REGION Network 4: Генерация аварии
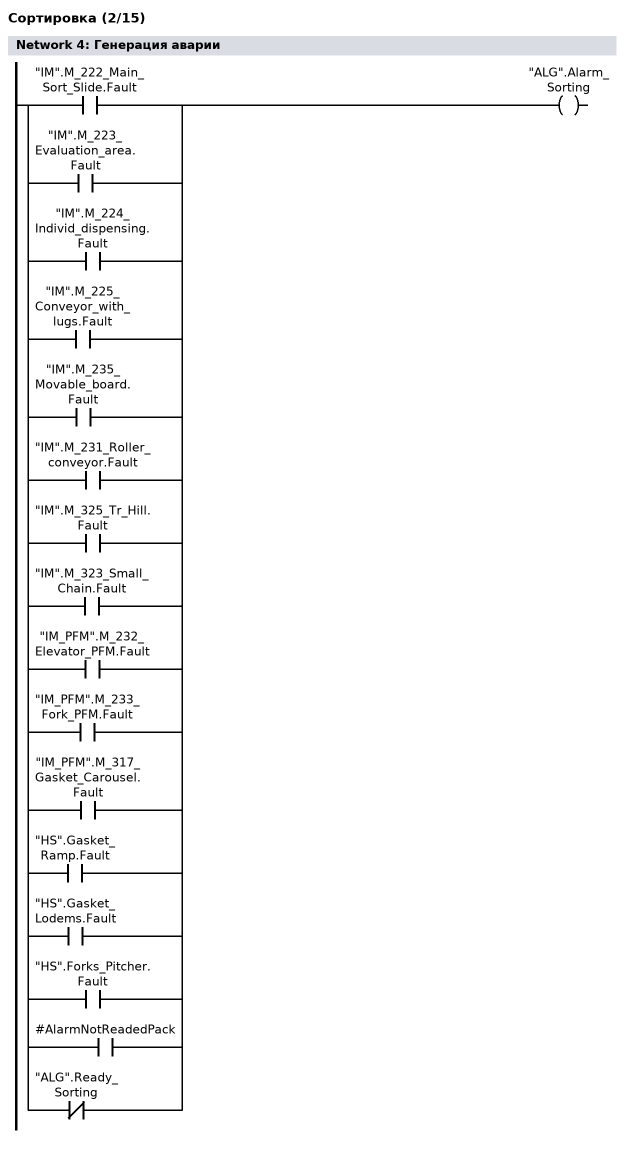
   RUNG wire#powerrail
      Contact( "IM".M_222_Main_Sort_Slide.Fault )
      wire#w1
      Coil( "ALG".Alarm_Sorting )
   END_RUNG
   RUNG wire#powerrail
      Contact( "IM".M_223_Evaluation_area.Fault )
   END_RUNG wire#w1
   RUNG wire#powerrail
      Contact( "IM".M_224_Individ_dispensing.Fault )
   END_RUNG wire#w1
   RUNG wire#powerrail
      Contact( "IM".M_225_Conveyor_with_lugs.Fault )
   END_RUNG wire#w1
   RUNG wire#powerrail
      Contact( "IM".M_235_Movable_board.Fault )
   END_RUNG wire#w1
   RUNG wire#powerrail
      Contact( "IM".M_231_Roller_conveyor.Fault )
   END_RUNG wire#w1
   RUNG wire#powerrail
      Contact( "IM".M_325_Tr_Hill.Fault )
   END_RUNG wire#w1
   RUNG wire#powerrail
      Contact( "IM".M_323_Small_Chain.Fault )
   END_RUNG wire#w1
   RUNG wire#powerrail
      Contact( "IM_PFM".M_232_Elevator_PFM.Fault )
   END_RUNG wire#w1
   RUNG wire#powerrail
      Contact( "IM_PFM".M_233_Fork_PFM.Fault )
   END_RUNG wire#w1
   RUNG wire#powerrail
      Contact( "IM_PFM".M_317_Gasket_Carousel.Fault )
   END_RUNG wire#w1
   RUNG wire#powerrail
      Contact( "HS".Gasket_Ramp.Fault )
   END_RUNG wire#w1
   RUNG wire#powerrail
      Contact( "HS".Gasket_Lodems.Fault )
   END_RUNG wire#w1
   RUNG wire#powerrail
      Contact( "HS".Forks_Pitcher.Fault )
   END_RUNG wire#w1
   RUNG wire#powerrail
      Contact( #AlarmNotReadedPack )
   END_RUNG wire#w1
   RUNG wire#powerrail
      I_Contact( "ALG".Ready_Sorting )
   END_RUNG wire#w1
   // the same network as SCL:
   "ALG".Alarm_Sorting := "IM".M_222_Main_Sort_Slide.Fault OR "IM".M_223_Evaluation_area.Fault OR "IM".M_224_Individ_dispensing.Fault OR "IM".M_225_Conveyor_with_lugs.Fault OR "IM".M_235_Movable_board.Fault OR "IM".M_231_Roller_conveyor.Fault OR "IM".M_325_Tr_Hill.Fault OR "IM".M_323_Small_Chain.Fault OR "IM_PFM".M_232_Elevator_PFM.Fault OR "IM_PFM".M_233_Fork_PFM.Fault OR "IM_PFM".M_317_Gasket_Carousel.Fault OR "HS".Gasket_Ramp.Fault OR "HS".Gasket_Lodems.Fault OR "HS".Forks_Pitcher.Fault OR #AlarmNotReadedPack OR NOT "ALG".Ready_Sorting;
END_REGION

REGION Network 5: Сбор аварий с других узлов + аварии не генерирующие останов линии
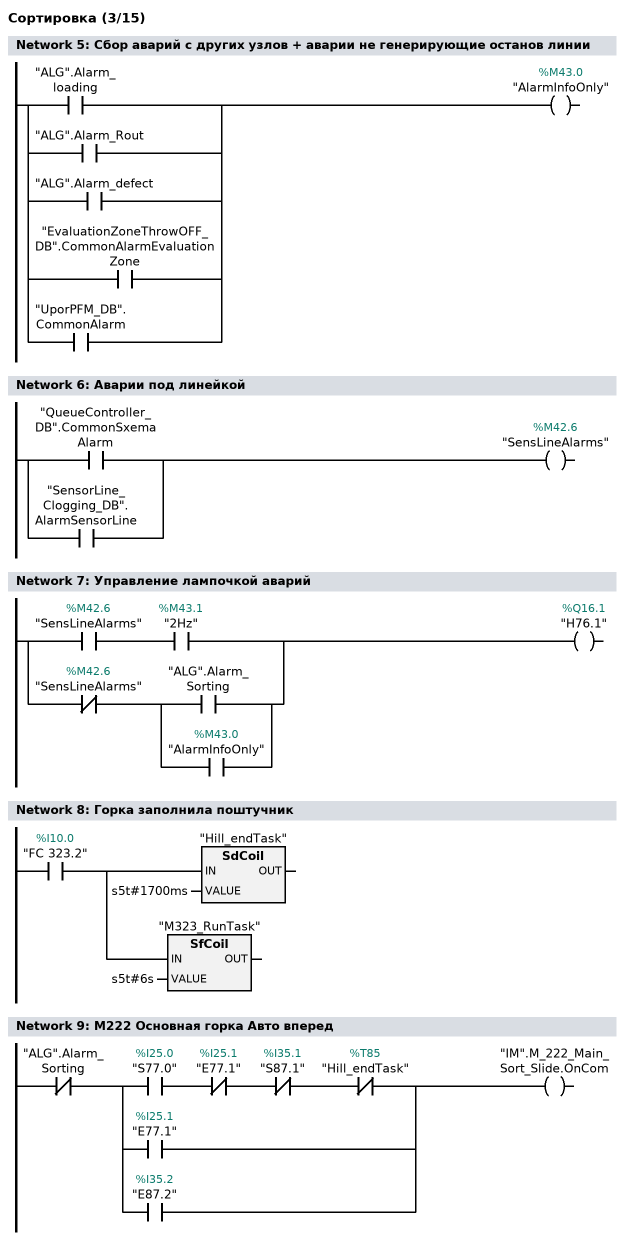
   RUNG wire#powerrail
      Contact( "ALG".Alarm_loading )
      wire#w1
      Coil( "AlarmInfoOnly" )
   END_RUNG
   RUNG wire#powerrail
      Contact( "ALG".Alarm_Rout )
   END_RUNG wire#w1
   RUNG wire#powerrail
      Contact( "ALG".Alarm_defect )
   END_RUNG wire#w1
   RUNG wire#powerrail
      Contact( "EvaluationZoneThrowOFF_DB".CommonAlarmEvaluationZone )
   END_RUNG wire#w1
   RUNG wire#powerrail
      Contact( "UporPFM_DB".CommonAlarm )
   END_RUNG wire#w1
   // the same network as SCL:
   "AlarmInfoOnly" := "ALG".Alarm_loading OR "ALG".Alarm_Rout OR "ALG".Alarm_defect OR "EvaluationZoneThrowOFF_DB".CommonAlarmEvaluationZone OR "UporPFM_DB".CommonAlarm;
END_REGION

REGION Network 6: Аварии под линейкой
   RUNG wire#powerrail
      Contact( "QueueController_DB".CommonSxemaAlarm )
      wire#w1
      Coil( "SensLineAlarms" )
   END_RUNG
   RUNG wire#powerrail
      Contact( "SensorLine_Clogging_DB".AlarmSensorLine )
   END_RUNG wire#w1
   // the same network as SCL:
   "SensLineAlarms" := "QueueController_DB".CommonSxemaAlarm OR "SensorLine_Clogging_DB".AlarmSensorLine;
END_REGION

REGION Network 7: Управление лампочкой аварий
   RUNG wire#powerrail
      Contact( "SensLineAlarms" )
      Contact( "2Hz" )
      wire#w1
      Coil( "H76.1" )
   END_RUNG
   RUNG wire#powerrail
      I_Contact( "SensLineAlarms" )
      wire#w2
      Contact( "ALG".Alarm_Sorting )
   END_RUNG wire#w1
   RUNG wire#w2
      Contact( "AlarmInfoOnly" )
   END_RUNG wire#w1
   // the same network as SCL:
   "H76.1" := ("SensLineAlarms" AND "2Hz") OR (NOT "SensLineAlarms" AND ("ALG".Alarm_Sorting OR "AlarmInfoOnly"));
END_REGION

REGION Network 8: Горка заполнила поштучник
   // no SCL statement known for SdCoil, SfCoil: written as a call
   #_w1 := "FC 323.2";
   SdCoil(in := "FC 323.2", value := s5t#1700ms, operand := "Hill_endTask");
   SfCoil(in := #_w1, value := s5t#6s, operand := "M323_RunTask");
END_REGION

REGION Network 9: М222 Основная горка Авто вперед
   RUNG wire#powerrail
      I_Contact( "ALG".Alarm_Sorting )
      wire#w1
      Contact( "S77.0" )
      I_Contact( "E77.1" )
      I_Contact( "S87.1" )
      I_Contact( "Hill_endTask" )
      wire#w2
      Coil( "IM".M_222_Main_Sort_Slide.OnCom )
   END_RUNG
   RUNG wire#w1
      Contact( "E77.1" )
   END_RUNG wire#w2
   RUNG wire#w1
      Contact( "E87.2" )
   END_RUNG wire#w2
   // the same network as SCL:
   "IM".M_222_Main_Sort_Slide.OnCom := NOT "ALG".Alarm_Sorting AND (("S77.0" AND NOT "E77.1" AND NOT "S87.1" AND NOT "Hill_endTask") OR "E77.1" OR "E87.2");
END_REGION

REGION Network 10: М222 Основная горка команда на движениее
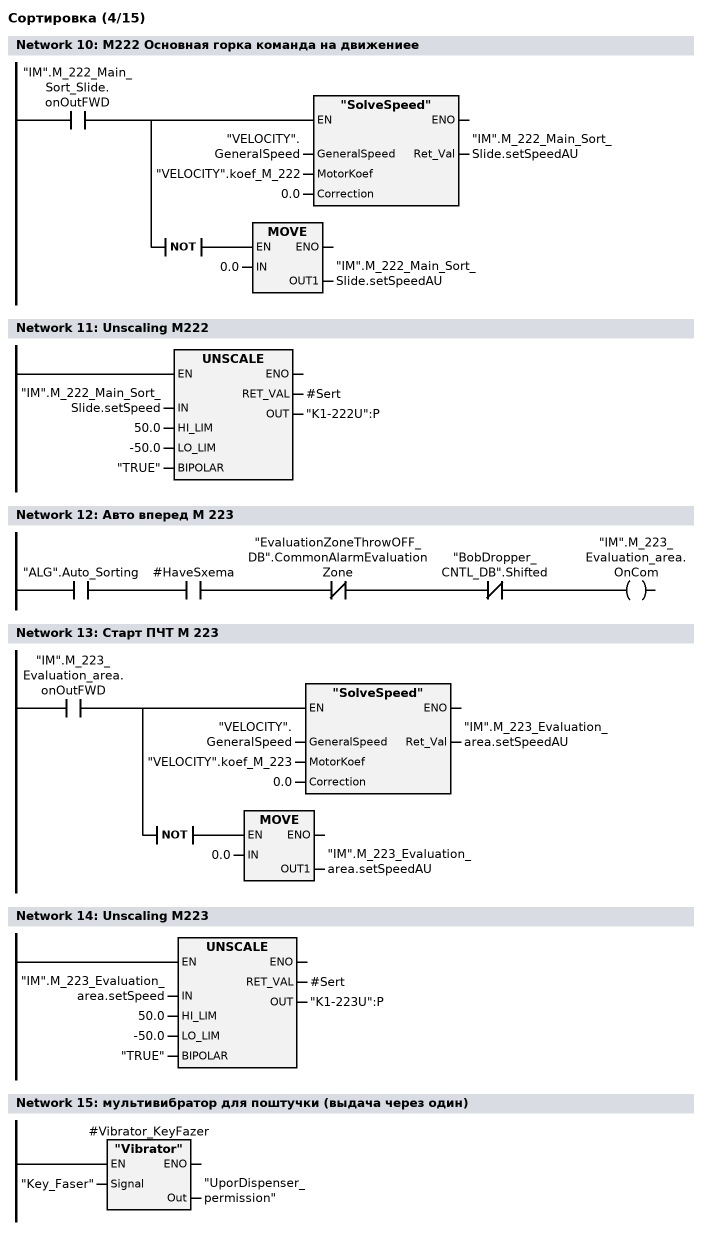
   RUNG wire#powerrail
      Contact( "IM".M_222_Main_Sort_Slide.onOutFWD )
      wire#w1
      "SolveSpeed"(GeneralSpeed := "VELOCITY".GeneralSpeed, MotorKoef := "VELOCITY".koef_M_222, Correction := 0.0, Ret_Val => "IM".M_222_Main_Sort_Slide.setSpeedAU)
   END_RUNG
   RUNG wire#w1
      Not()
      { S7_GenerateENO := "TRUE" } Move(in := 0.0, out1 => "IM".M_222_Main_Sort_Slide.setSpeedAU)
   END_RUNG
   // the same network as SCL:
   #_w1 := "IM".M_222_Main_Sort_Slide.onOutFWD;
   IF #_w1 THEN
       "IM".M_222_Main_Sort_Slide.setSpeedAU := "SolveSpeed"(GeneralSpeed := "VELOCITY".GeneralSpeed,
                               MotorKoef := "VELOCITY".koef_M_222,
                               Correction := 0.0);
   END_IF;
   IF NOT #_w1 THEN "IM".M_222_Main_Sort_Slide.setSpeedAU := 0.0; END_IF;
END_REGION

REGION Network 11: Unscaling M222
   RUNG wire#powerrail
      UNSCALE(IN := "IM".M_222_Main_Sort_Slide.setSpeed, HI_LIM := 50.0, LO_LIM := -50.0, BIPOLAR := "TRUE", RET_VAL => #Sert, OUT => "K1-222U":P)
   END_RUNG
   // the same network as SCL:
   #Sert := UNSCALE(IN := "IM".M_222_Main_Sort_Slide.setSpeed,
                    HI_LIM := 50.0,
                    LO_LIM := -50.0,
                    BIPOLAR := "TRUE",
                    OUT => "K1-222U":P);
END_REGION

REGION Network 12: Авто вперед M 223
   RUNG wire#powerrail
      Contact( "ALG".Auto_Sorting )
      Contact( #HaveSxema )
      I_Contact( "EvaluationZoneThrowOFF_DB".CommonAlarmEvaluationZone )
      I_Contact( "BobDropper_CNTL_DB".Shifted )
      Coil( "IM".M_223_Evaluation_area.OnCom )
   END_RUNG
   // the same network as SCL:
   "IM".M_223_Evaluation_area.OnCom := "ALG".Auto_Sorting AND #HaveSxema AND NOT "EvaluationZoneThrowOFF_DB".CommonAlarmEvaluationZone AND NOT "BobDropper_CNTL_DB".Shifted;
END_REGION

REGION Network 13: Старт ПЧТ М 223
   RUNG wire#powerrail
      Contact( "IM".M_223_Evaluation_area.onOutFWD )
      wire#w1
      "SolveSpeed"(GeneralSpeed := "VELOCITY".GeneralSpeed, MotorKoef := "VELOCITY".koef_M_223, Correction := 0.0, Ret_Val => "IM".M_223_Evaluation_area.setSpeedAU)
   END_RUNG
   RUNG wire#w1
      Not()
      { S7_GenerateENO := "TRUE" } Move(in := 0.0, out1 => "IM".M_223_Evaluation_area.setSpeedAU)
   END_RUNG
   // the same network as SCL:
   #_w1 := "IM".M_223_Evaluation_area.onOutFWD;
   IF #_w1 THEN
       "IM".M_223_Evaluation_area.setSpeedAU := "SolveSpeed"(GeneralSpeed := "VELOCITY".GeneralSpeed,
                               MotorKoef := "VELOCITY".koef_M_223,
                               Correction := 0.0);
   END_IF;
   IF NOT #_w1 THEN "IM".M_223_Evaluation_area.setSpeedAU := 0.0; END_IF;
END_REGION

REGION Network 14: Unscaling M223
   RUNG wire#powerrail
      UNSCALE(IN := "IM".M_223_Evaluation_area.setSpeed, HI_LIM := 50.0, LO_LIM := -50.0, BIPOLAR := "TRUE", RET_VAL => #Sert, OUT => "K1-223U":P)
   END_RUNG
   // the same network as SCL:
   #Sert := UNSCALE(IN := "IM".M_223_Evaluation_area.setSpeed,
                    HI_LIM := 50.0,
                    LO_LIM := -50.0,
                    BIPOLAR := "TRUE",
                    OUT => "K1-223U":P);
END_REGION

REGION Network 15: мультивибратор для поштучки (выдача через один)
   RUNG wire#powerrail
      #Vibrator_KeyFazer(Signal := "Key_Faser", Out => "UporDispenser_permission")
   END_RUNG
   // the same network as SCL:
   #Vibrator_KeyFazer(Signal := "Key_Faser", Out => "UporDispenser_permission");   // "Vibrator"
END_REGION

REGION Network 16: Есть схема для сортировки
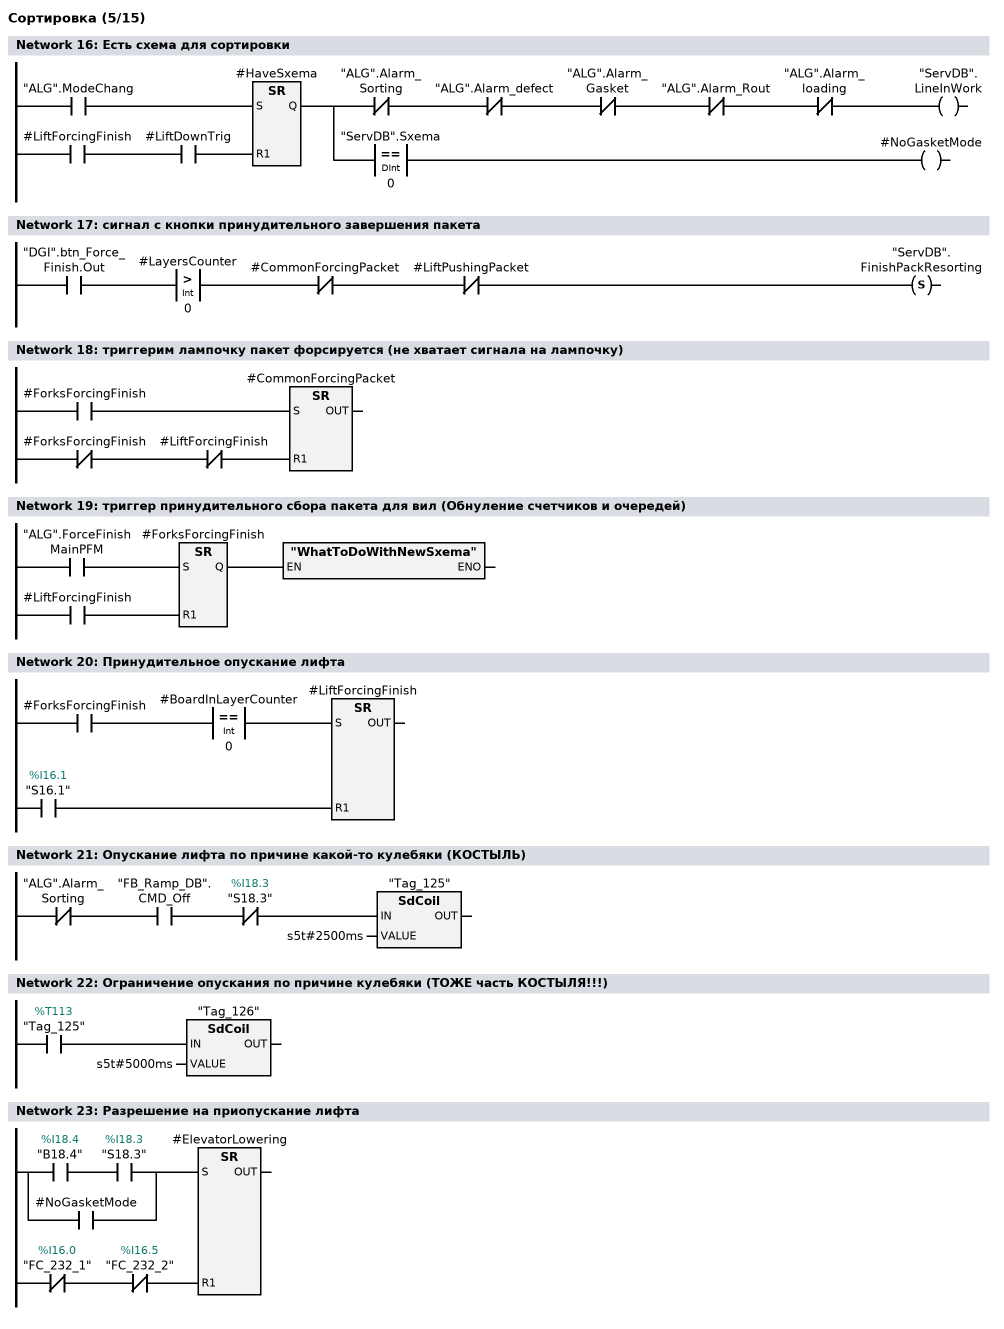
   RUNG wire#powerrail
      Contact( "ALG".ModeChang )
      S_SR(operand := #HaveSxema, r1 := wire#w1)
      wire#w2
      I_Contact( "ALG".Alarm_Sorting )
      I_Contact( "ALG".Alarm_defect )
      I_Contact( "ALG".Alarm_Gasket )
      I_Contact( "ALG".Alarm_Rout )
      I_Contact( "ALG".Alarm_loading )
      Coil( "ServDB".LineInWork )
   END_RUNG
   RUNG wire#powerrail
      Contact( #LiftForcingFinish )
      Contact( #LiftDownTrig )
   END_RUNG wire#w1
   RUNG wire#w2
      { S7_Templates := "SrcType := DInt" } EQ_Contact(in1 := "ServDB".Sxema, in2 := 0)
      Coil( #NoGasketMode )
   END_RUNG
   // the same network as SCL:
   IF "ALG".ModeChang THEN
       #HaveSxema := TRUE;   // SR flip-flop
   END_IF;
   IF #LiftForcingFinish AND #LiftDownTrig THEN #HaveSxema := FALSE; END_IF;
   "ServDB".LineInWork := #HaveSxema AND NOT "ALG".Alarm_Sorting AND NOT "ALG".Alarm_defect AND NOT "ALG".Alarm_Gasket AND NOT "ALG".Alarm_Rout AND NOT "ALG".Alarm_loading;
   #NoGasketMode := #HaveSxema AND ("ServDB".Sxema = 0);
END_REGION

REGION Network 17: сигнал с кнопки принудительного завершения пакета
   RUNG wire#powerrail
      Contact( "DGI".btn_Force_Finish.Out )
      { S7_Templates := "SrcType := Int" } GT_Contact(in1 := #LayersCounter, in2 := 0)
      I_Contact( #CommonForcingPacket )
      I_Contact( #LiftPushingPacket )
      S_Coil( "ServDB".FinishPackResorting )
   END_RUNG
   // the same network as SCL:
   IF "DGI".btn_Force_Finish.Out AND (#LayersCounter > 0) AND NOT #CommonForcingPacket AND NOT #LiftPushingPacket THEN
       "ServDB".FinishPackResorting := TRUE;
   END_IF;
END_REGION

REGION Network 18: триггерим лампочку пакет форсируется (не хватает сигнала на лампочку)
   RUNG wire#powerrail
      Contact( #ForksForcingFinish )
      S_SR(operand := #CommonForcingPacket, r1 := wire#w1)
   END_RUNG
   RUNG wire#powerrail
      I_Contact( #ForksForcingFinish )
      I_Contact( #LiftForcingFinish )
   END_RUNG wire#w1
   // the same network as SCL:
   IF #ForksForcingFinish THEN
       #CommonForcingPacket := TRUE;   // SR flip-flop
   END_IF;
   IF NOT #ForksForcingFinish AND NOT #LiftForcingFinish THEN #CommonForcingPacket := FALSE; END_IF;
END_REGION

REGION Network 19: триггер принудительного сбора пакета для вил (Обнуление счетчиков и очередей)
   RUNG wire#powerrail
      Contact( "ALG".ForceFinishMainPFM )
      S_SR(operand := #ForksForcingFinish, r1 := wire#w1)
      "WhatToDoWithNewSxema"()
   END_RUNG
   RUNG wire#powerrail
      Contact( #LiftForcingFinish )
   END_RUNG wire#w1
   // the same network as SCL:
   IF "ALG".ForceFinishMainPFM THEN
       #ForksForcingFinish := TRUE;   // SR flip-flop
   END_IF;
   IF #LiftForcingFinish THEN #ForksForcingFinish := FALSE; END_IF;
   IF #ForksForcingFinish THEN "WhatToDoWithNewSxema"(); END_IF;
END_REGION

REGION Network 20: Принудительное опускание лифта
   RUNG wire#powerrail
      Contact( #ForksForcingFinish )
      { S7_Templates := "SrcType := Int" } EQ_Contact(in1 := #BoardInLayerCounter, in2 := 0)
      S_SR(operand := #LiftForcingFinish, r1 := wire#w1)
   END_RUNG
   RUNG wire#powerrail
      Contact( "S16.1" )
   END_RUNG wire#w1
   // the same network as SCL:
   IF #ForksForcingFinish AND (#BoardInLayerCounter = 0) THEN
       #LiftForcingFinish := TRUE;   // SR flip-flop
   END_IF;
   IF "S16.1" THEN #LiftForcingFinish := FALSE; END_IF;
END_REGION

REGION Network 21: Опускание лифта по причине какой-то кулебяки (КОСТЫЛЬ)
   // no SCL statement known for SdCoil: written as a call
   SdCoil(in := NOT "ALG".Alarm_Sorting AND "FB_Ramp_DB".CMD_Off AND NOT "S18.3",
          value := s5t#2500ms,
          operand := "Tag_125");
END_REGION

REGION Network 22: Ограничение опускания по причине кулебяки (ТОЖЕ часть КОСТЫЛЯ!!!)
   // no SCL statement known for SdCoil: written as a call
   SdCoil(in := "Tag_125", value := s5t#5000ms, operand := "Tag_126");
END_REGION

REGION Network 23: Разрешение на приопускание лифта
   RUNG wire#powerrail
      Contact( "B18.4" )
      Contact( "S18.3" )
      wire#w1
      S_SR(operand := #ElevatorLowering, r1 := wire#w2)
   END_RUNG
   RUNG wire#powerrail
      Contact( #NoGasketMode )
   END_RUNG wire#w1
   RUNG wire#powerrail
      I_Contact( "FC_232_1" )
      I_Contact( "FC_232_2" )
   END_RUNG wire#w2
   // the same network as SCL:
   IF ("B18.4" AND "S18.3") OR #NoGasketMode THEN
       #ElevatorLowering := TRUE;   // SR flip-flop
   END_IF;
   IF NOT "FC_232_1" AND NOT "FC_232_2" THEN #ElevatorLowering := FALSE; END_IF;
END_REGION

REGION Network 24: Счёт слоёв
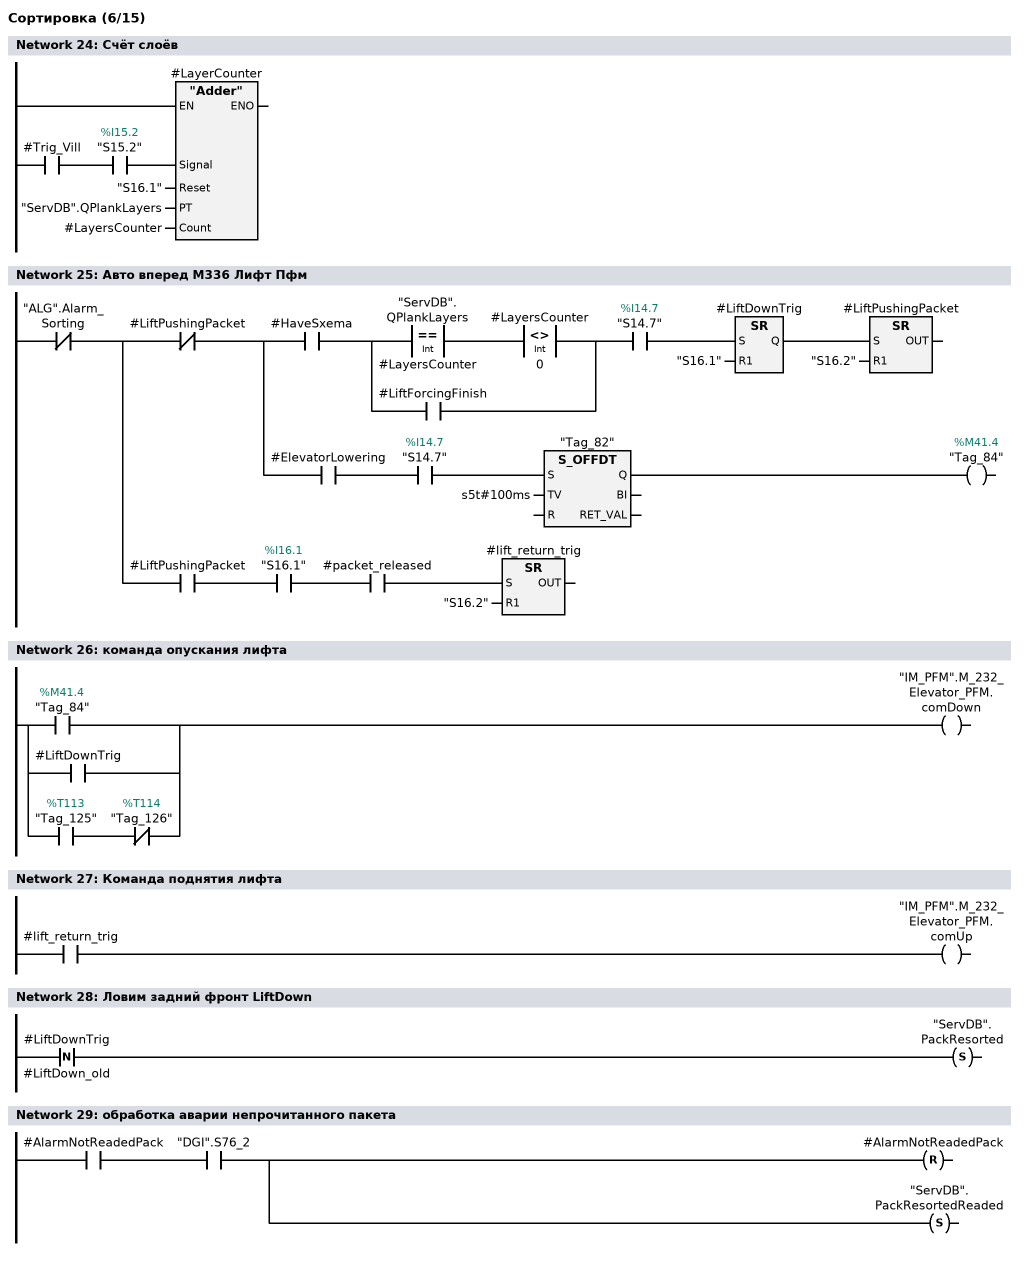
   RUNG wire#powerrail
      #LayerCounter(Signal := wire#w1, Reset := "S16.1", PT := "ServDB".QPlankLayers, Count := #LayersCounter)
   END_RUNG
   RUNG wire#powerrail
      Contact( #Trig_Vill )
      Contact( "S15.2" )
   END_RUNG wire#w1
   // the same network as SCL:
   #LayerCounter(Signal := #Trig_Vill AND "S15.2",   // "Adder"
                 Reset := "S16.1",
                 PT := "ServDB".QPlankLayers,
                 Count := #LayersCounter);
END_REGION

REGION Network 25: Авто вперед М336 Лифт Пфм
   RUNG wire#powerrail
      I_Contact( "ALG".Alarm_Sorting )
      wire#w1
      I_Contact( #LiftPushingPacket )
      wire#w2
      Contact( #HaveSxema )
      wire#w3
      { S7_Templates := "SrcType := Int" } EQ_Contact(in1 := "ServDB".QPlankLayers, in2 := #LayersCounter)
      { S7_Templates := "SrcType := Int" } NE_Contact(in1 := #LayersCounter, in2 := 0)
      wire#w4
      Contact( "S14.7" )
      S_SR(operand := #LiftDownTrig, r1 := "S16.1")
      S_SR(operand := #LiftPushingPacket, r1 := "S16.2")
   END_RUNG
   RUNG wire#w3
      Contact( #LiftForcingFinish )
   END_RUNG wire#w4
   RUNG wire#w2
      Contact( #ElevatorLowering )
      Contact( "S14.7" )
      S_OFFDT(T_NO := "Tag_82", TV := s5t#100ms, R :=, BI =>, RET_VAL =>)
      Coil( "Tag_84" )
   END_RUNG
   RUNG wire#w1
      Contact( #LiftPushingPacket )
      Contact( "S16.1" )
      Contact( #packet_released )
      S_SR(operand := #lift_return_trig, r1 := "S16.2")
   END_RUNG
   // the same network as SCL:
   #_w1 := NOT "ALG".Alarm_Sorting AND NOT #LiftPushingPacket;
   IF #_w1 AND #HaveSxema AND ((("ServDB".QPlankLayers = #LayersCounter) AND (#LayersCounter <> 0)) OR #LiftForcingFinish) AND "S14.7" THEN
       #LiftDownTrig := TRUE;   // SR flip-flop
   END_IF;
   IF "S16.1" THEN #LiftDownTrig := FALSE; END_IF;
   IF #LiftDownTrig THEN
       #LiftPushingPacket := TRUE;   // SR flip-flop
   END_IF;
   IF "S16.2" THEN #LiftPushingPacket := FALSE; END_IF;
   #_s5time1 := S_OFFDT(T_NO := "Tag_82",
                        S := #_w1 AND #ElevatorLowering AND "S14.7",
                        TV := s5t#100ms,
                        Q => #_w2);
   "Tag_84" := #_w2;
   IF NOT "ALG".Alarm_Sorting AND #LiftPushingPacket AND "S16.1" AND #packet_released THEN
       #lift_return_trig := TRUE;   // SR flip-flop
   END_IF;
   IF "S16.2" THEN #lift_return_trig := FALSE; END_IF;
END_REGION

REGION Network 26: команда опускания лифта
   RUNG wire#powerrail
      Contact( "Tag_84" )
      wire#w1
      Coil( "IM_PFM".M_232_Elevator_PFM.comDown )
   END_RUNG
   RUNG wire#powerrail
      Contact( #LiftDownTrig )
   END_RUNG wire#w1
   RUNG wire#powerrail
      Contact( "Tag_125" )
      I_Contact( "Tag_126" )
   END_RUNG wire#w1
   // the same network as SCL:
   "IM_PFM".M_232_Elevator_PFM.comDown := "Tag_84" OR #LiftDownTrig OR ("Tag_125" AND NOT "Tag_126");
END_REGION

REGION Network 27: Команда поднятия лифта
   RUNG wire#powerrail
      Contact( #lift_return_trig )
      Coil( "IM_PFM".M_232_Elevator_PFM.comUp )
   END_RUNG
   // the same network as SCL:
   "IM_PFM".M_232_Elevator_PFM.comUp := #lift_return_trig;
END_REGION

REGION Network 28: Ловим задний фронт LiftDown
   RUNG wire#powerrail
      N_Contact(operand := #LiftDownTrig, bit := #LiftDown_old)
      S_Coil( "ServDB".PackResorted )
   END_RUNG
   // the same network as SCL:
   #_w1 := NOT #LiftDownTrig AND #LiftDown_old;   // falling edge of #LiftDownTrig
   #LiftDown_old := #LiftDownTrig;
   IF #_w1 THEN "ServDB".PackResorted := TRUE; END_IF;
END_REGION

REGION Network 29: обработка аварии непрочитанного пакета
   RUNG wire#powerrail
      Contact( #AlarmNotReadedPack )
      Contact( "DGI".S76_2 )
      wire#w1
      R_Coil( #AlarmNotReadedPack )
   END_RUNG
   RUNG wire#w1
      S_Coil( "ServDB".PackResortedReaded )
   END_RUNG
   // the same network as SCL:
   #_w1 := #AlarmNotReadedPack AND "DGI".S76_2;
   IF #_w1 THEN
       #AlarmNotReadedPack := FALSE;
       "ServDB".PackResortedReaded := TRUE;
   END_IF;
END_REGION

REGION Network 30: Ловим задний фронт LiftPushing
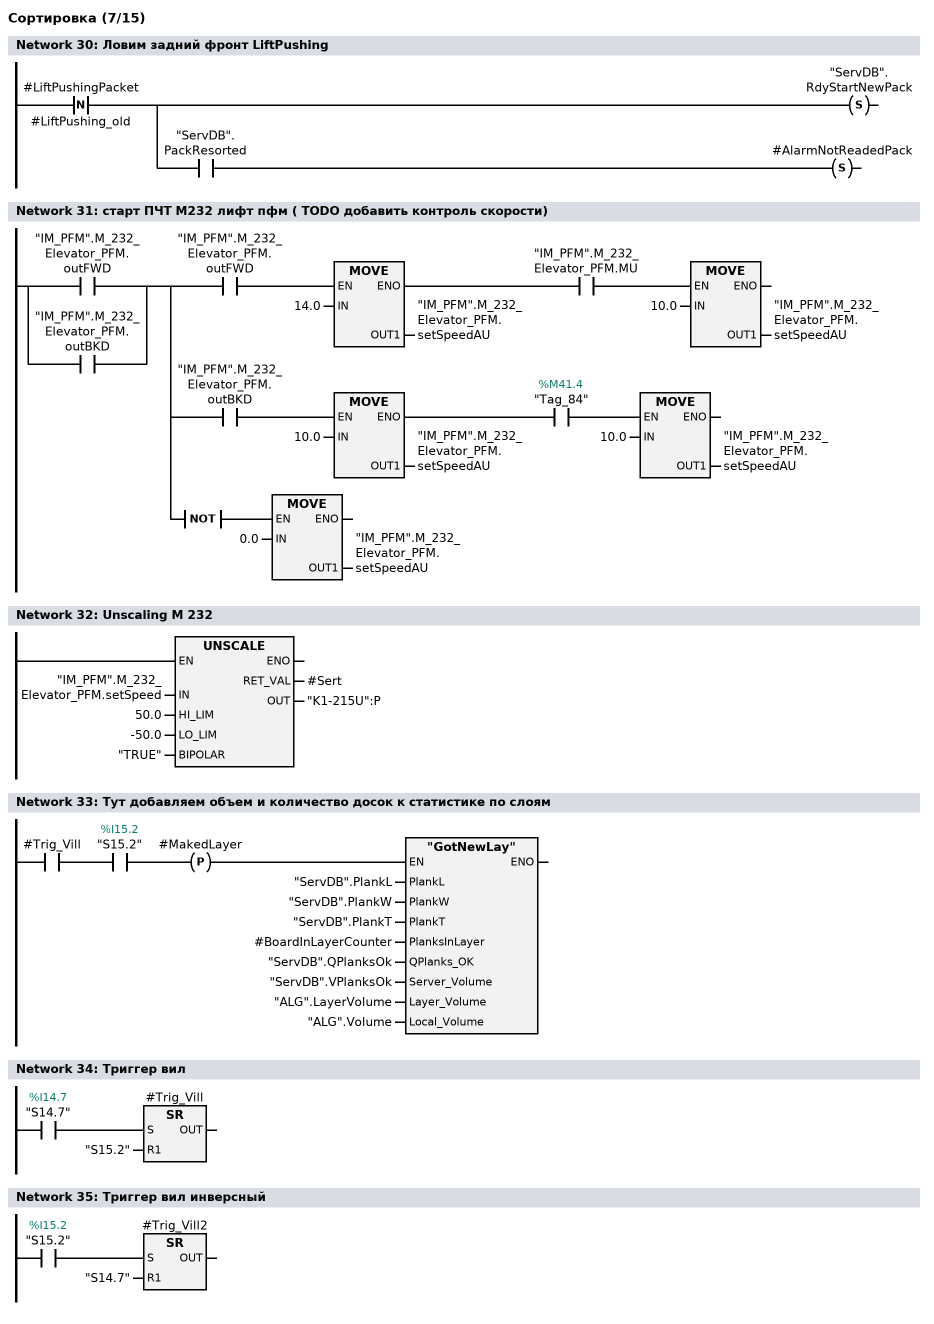
   RUNG wire#powerrail
      N_Contact(operand := #LiftPushingPacket, bit := #LiftPushing_old)
      wire#w1
      S_Coil( "ServDB".RdyStartNewPack )
   END_RUNG
   RUNG wire#w1
      Contact( "ServDB".PackResorted )
      S_Coil( #AlarmNotReadedPack )
   END_RUNG
   // the same network as SCL:
   #_w1 := NOT #LiftPushingPacket AND #LiftPushing_old;   // falling edge of #LiftPushingPacket
   #LiftPushing_old := #LiftPushingPacket;
   IF #_w1 THEN "ServDB".RdyStartNewPack := TRUE; END_IF;
   IF #_w1 AND "ServDB".PackResorted THEN #AlarmNotReadedPack := TRUE; END_IF;
END_REGION

REGION Network 31: старт ПЧТ М232 лифт пфм ( TODO добавить контроль скорости)
   RUNG wire#powerrail
      Contact( "IM_PFM".M_232_Elevator_PFM.outFWD )
      wire#w1
      Contact( "IM_PFM".M_232_Elevator_PFM.outFWD )
      { S7_GenerateENO := "TRUE" } Move(in := 14.0, out1 => "IM_PFM".M_232_Elevator_PFM.setSpeedAU)
      Contact( "IM_PFM".M_232_Elevator_PFM.MU )
      { S7_GenerateENO := "TRUE" } Move(in := 10.0, out1 => "IM_PFM".M_232_Elevator_PFM.setSpeedAU)
   END_RUNG
   RUNG wire#powerrail
      Contact( "IM_PFM".M_232_Elevator_PFM.outBKD )
   END_RUNG wire#w1
   RUNG wire#w1
      Contact( "IM_PFM".M_232_Elevator_PFM.outBKD )
      { S7_GenerateENO := "TRUE" } Move(in := 10.0, out1 => "IM_PFM".M_232_Elevator_PFM.setSpeedAU)
      Contact( "Tag_84" )
      { S7_GenerateENO := "TRUE" } Move(in := 10.0, out1 => "IM_PFM".M_232_Elevator_PFM.setSpeedAU)
   END_RUNG
   RUNG wire#w1
      Not()
      { S7_GenerateENO := "TRUE" } Move(in := 0.0, out1 => "IM_PFM".M_232_Elevator_PFM.setSpeedAU)
   END_RUNG
   // the same network as SCL:
   // ENO of a box is taken as its EN; it also drops when the box reports an error
   #_w1 := "IM_PFM".M_232_Elevator_PFM.outFWD OR "IM_PFM".M_232_Elevator_PFM.outBKD;
   #_w2 := #_w1 AND "IM_PFM".M_232_Elevator_PFM.outFWD;
   IF #_w2 THEN "IM_PFM".M_232_Elevator_PFM.setSpeedAU := 14.0; END_IF;
   IF #_w2 AND "IM_PFM".M_232_Elevator_PFM.MU THEN "IM_PFM".M_232_Elevator_PFM.setSpeedAU := 10.0; END_IF;
   #_w3 := #_w1 AND "IM_PFM".M_232_Elevator_PFM.outBKD;
   IF #_w3 THEN "IM_PFM".M_232_Elevator_PFM.setSpeedAU := 10.0; END_IF;
   IF #_w3 AND "Tag_84" THEN "IM_PFM".M_232_Elevator_PFM.setSpeedAU := 10.0; END_IF;
   IF NOT #_w1 THEN "IM_PFM".M_232_Elevator_PFM.setSpeedAU := 0.0; END_IF;
END_REGION

REGION Network 32: Unscaling M 232
   RUNG wire#powerrail
      UNSCALE(IN := "IM_PFM".M_232_Elevator_PFM.setSpeed, HI_LIM := 50.0, LO_LIM := -50.0, BIPOLAR := "TRUE", RET_VAL => #Sert, OUT => "K1-215U":P)
   END_RUNG
   // the same network as SCL:
   #Sert := UNSCALE(IN := "IM_PFM".M_232_Elevator_PFM.setSpeed,
                    HI_LIM := 50.0,
                    LO_LIM := -50.0,
                    BIPOLAR := "TRUE",
                    OUT => "K1-215U":P);
END_REGION

REGION Network 33: Тут добавляем объем и количество досок к статистике по слоям
   RUNG wire#powerrail
      Contact( #Trig_Vill )
      Contact( "S15.2" )
      P_Trig( #MakedLayer )
      "GotNewLay"(PlankL := "ServDB".PlankL, PlankW := "ServDB".PlankW, PlankT := "ServDB".PlankT, PlanksInLayer := #BoardInLayerCounter, QPlanks_OK := "ServDB".QPlanksOk, Server_Volume := "ServDB".VPlanksOk, Layer_Volume := "ALG".LayerVolume, Local_Volume := "ALG".Volume)
   END_RUNG
   // the same network as SCL:
   #_w1 := #Trig_Vill AND "S15.2";
   #_w2 := #_w1 AND NOT #MakedLayer;   // rising edge
   #MakedLayer := #_w1;
   IF #_w2 THEN
       "GotNewLay"(PlankL := "ServDB".PlankL,
                   PlankW := "ServDB".PlankW,
                   PlankT := "ServDB".PlankT,
                   PlanksInLayer := #BoardInLayerCounter,
                   QPlanks_OK := "ServDB".QPlanksOk,
                   Server_Volume := "ServDB".VPlanksOk,
                   Layer_Volume := "ALG".LayerVolume,
                   Local_Volume := "ALG".Volume);
   END_IF;
END_REGION

REGION Network 34: Триггер вил
   RUNG wire#powerrail
      Contact( "S14.7" )
      S_SR(operand := #Trig_Vill, r1 := "S15.2")
   END_RUNG
   // the same network as SCL:
   IF "S14.7" THEN
       #Trig_Vill := TRUE;   // SR flip-flop
   END_IF;
   IF "S15.2" THEN #Trig_Vill := FALSE; END_IF;
END_REGION

REGION Network 35: Триггер вил инверсный
   RUNG wire#powerrail
      Contact( "S15.2" )
      S_SR(operand := #Trig_Vill2, r1 := "S14.7")
   END_RUNG
   // the same network as SCL:
   IF "S15.2" THEN
       #Trig_Vill2 := TRUE;   // SR flip-flop
   END_IF;
   IF "S14.7" THEN #Trig_Vill2 := FALSE; END_IF;
END_REGION

REGION Network 36: Контроль кейфазеров на М225 и Счет досок на слой ПФМ (Счет не вызываем)
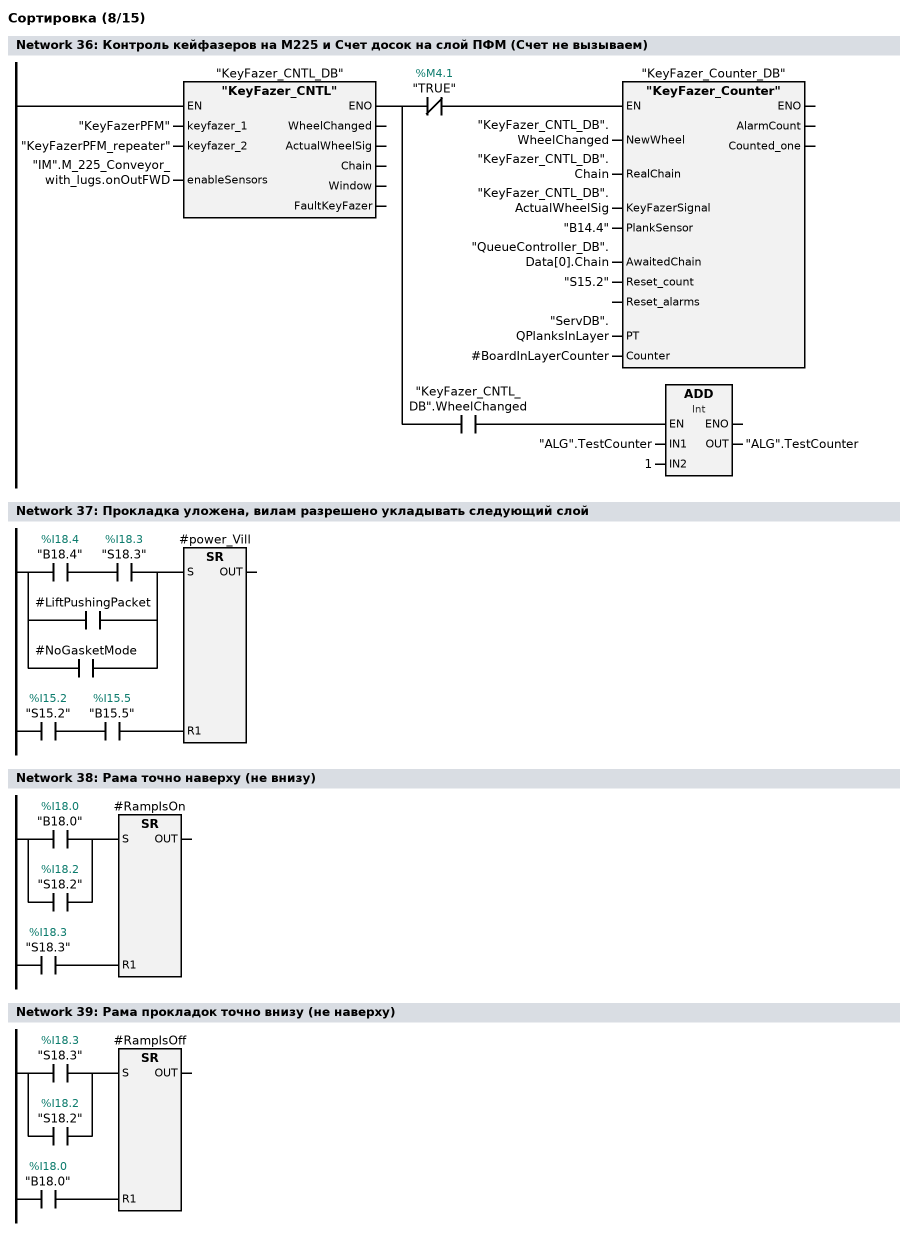
   RUNG wire#powerrail
      "KeyFazer_CNTL_DB"(keyfazer_1 := "KeyFazerPFM", keyfazer_2 := "KeyFazerPFM_repeater", enableSensors := "IM".M_225_Conveyor_with_lugs.onOutFWD, WheelChanged =>, ActualWheelSig =>, Chain =>, Window =>, FaultKeyFazer =>)
      wire#w1
      I_Contact( "TRUE" )
      "KeyFazer_Counter_DB"(NewWheel := "KeyFazer_CNTL_DB".WheelChanged, RealChain := "KeyFazer_CNTL_DB".Chain, KeyFazerSignal := "KeyFazer_CNTL_DB".ActualWheelSig, PlankSensor := "B14.4", AwaitedChain := "QueueController_DB".Data[0].Chain, Reset_count := "S15.2", Reset_alarms :=, PT := "ServDB".QPlanksInLayer, "Counter" := #BoardInLayerCounter, AlarmCount =>, Counted_one =>)
   END_RUNG
   RUNG wire#w1
      Contact( "KeyFazer_CNTL_DB".WheelChanged )
      { S7_Templates := "SrcType := Int"; S7_GenerateENO := "TRUE" } Add(in1 := "ALG".TestCounter, in2 := 1, out => "ALG".TestCounter)
   END_RUNG
   // the same network as SCL:
   "KeyFazer_CNTL_DB"(keyfazer_1 := "KeyFazerPFM",   // "KeyFazer_CNTL"
                      keyfazer_2 := "KeyFazerPFM_repeater",
                      enableSensors := "IM".M_225_Conveyor_with_lugs.onOutFWD,
                      ENO => #_w1);
   IF #_w1 AND NOT "TRUE" THEN
       "KeyFazer_Counter_DB"(NewWheel := "KeyFazer_CNTL_DB".WheelChanged,   // "KeyFazer_Counter"
                             RealChain := "KeyFazer_CNTL_DB".Chain,
                             KeyFazerSignal := "KeyFazer_CNTL_DB".ActualWheelSig,
                             PlankSensor := "B14.4",
                             AwaitedChain := "QueueController_DB".Data[0].Chain,
                             Reset_count := "S15.2",
                             PT := "ServDB".QPlanksInLayer,
                             "Counter" := #BoardInLayerCounter);
   END_IF;
   IF #_w1 AND "KeyFazer_CNTL_DB".WheelChanged THEN "ALG".TestCounter := "ALG".TestCounter + 1; END_IF;
END_REGION

REGION Network 37: Прокладка уложена, вилам разрешено укладывать следующий слой
   RUNG wire#powerrail
      Contact( "B18.4" )
      Contact( "S18.3" )
      wire#w1
      S_SR(operand := #power_Vill, r1 := wire#w2)
   END_RUNG
   RUNG wire#powerrail
      Contact( #LiftPushingPacket )
   END_RUNG wire#w1
   RUNG wire#powerrail
      Contact( #NoGasketMode )
   END_RUNG wire#w1
   RUNG wire#powerrail
      Contact( "S15.2" )
      Contact( "B15.5" )
   END_RUNG wire#w2
   // the same network as SCL:
   IF ("B18.4" AND "S18.3") OR #LiftPushingPacket OR #NoGasketMode THEN
       #power_Vill := TRUE;   // SR flip-flop
   END_IF;
   IF "S15.2" AND "B15.5" THEN #power_Vill := FALSE; END_IF;
END_REGION

REGION Network 38: Рама точно наверху (не внизу)
   RUNG wire#powerrail
      Contact( "B18.0" )
      wire#w1
      S_SR(operand := #RampIsOn, r1 := wire#w2)
   END_RUNG
   RUNG wire#powerrail
      Contact( "S18.2" )
   END_RUNG wire#w1
   RUNG wire#powerrail
      Contact( "S18.3" )
   END_RUNG wire#w2
   // the same network as SCL:
   IF "B18.0" OR "S18.2" THEN
       #RampIsOn := TRUE;   // SR flip-flop
   END_IF;
   IF "S18.3" THEN #RampIsOn := FALSE; END_IF;
END_REGION

REGION Network 39: Рама прокладок точно внизу (не наверху)
   RUNG wire#powerrail
      Contact( "S18.3" )
      wire#w1
      S_SR(operand := #RampIsOff, r1 := wire#w2)
   END_RUNG
   RUNG wire#powerrail
      Contact( "S18.2" )
   END_RUNG wire#w1
   RUNG wire#powerrail
      Contact( "B18.0" )
   END_RUNG wire#w2
   // the same network as SCL:
   IF "S18.3" OR "S18.2" THEN
       #RampIsOff := TRUE;   // SR flip-flop
   END_IF;
   IF "B18.0" THEN #RampIsOff := FALSE; END_IF;
END_REGION

REGION Network 40: M 233 вилы авто
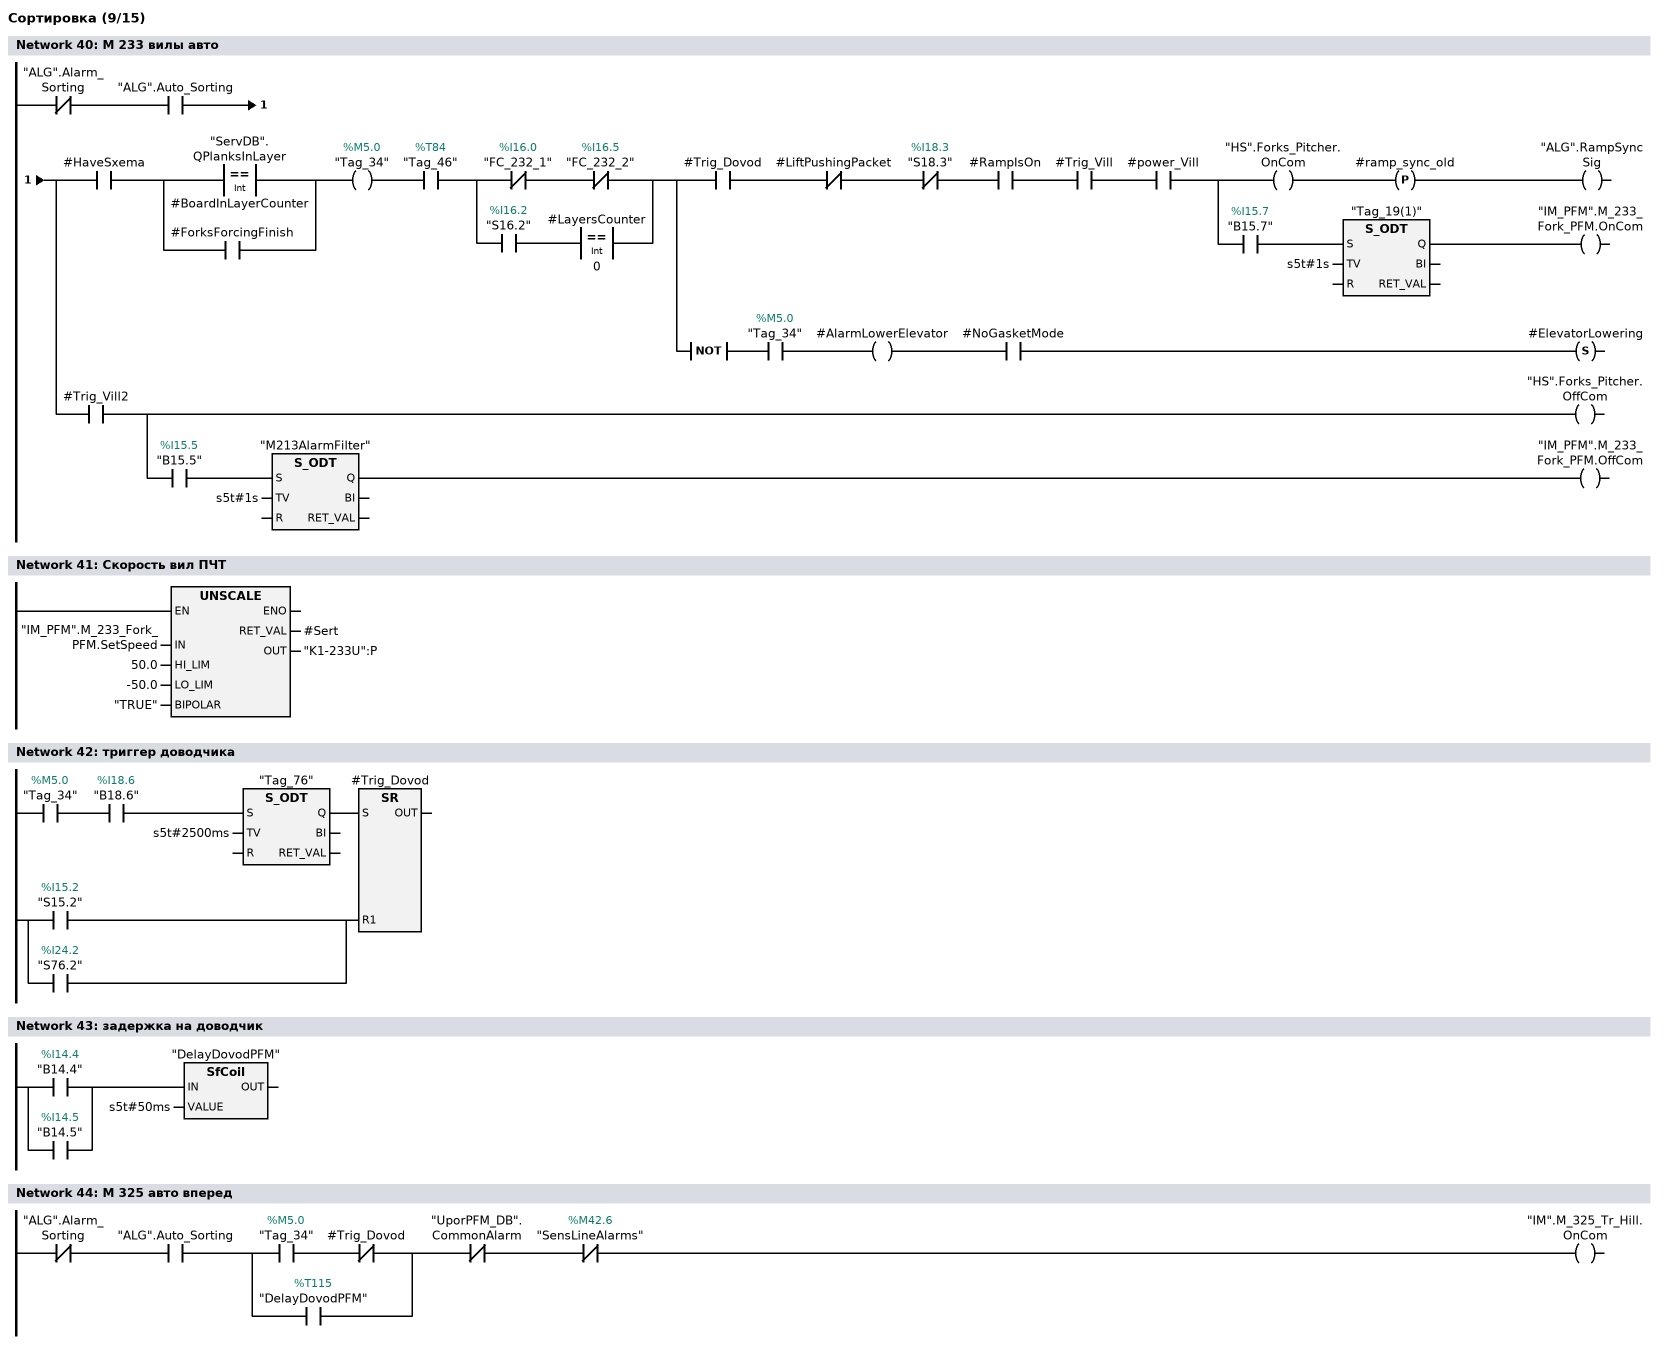
   RUNG wire#powerrail
      I_Contact( "ALG".Alarm_Sorting )
      Contact( "ALG".Auto_Sorting )
      wire#w1
      Contact( #HaveSxema )
      wire#w2
      { S7_Templates := "SrcType := Int" } EQ_Contact(in1 := "ServDB".QPlanksInLayer, in2 := #BoardInLayerCounter)
      wire#w3
      Coil( "Tag_34" )
      Contact( "Tag_46" )
      wire#w4
      I_Contact( "FC_232_1" )
      I_Contact( "FC_232_2" )
      wire#w5
      Contact( #Trig_Dovod )
      I_Contact( #LiftPushingPacket )
      I_Contact( "S18.3" )
      Contact( #RampIsOn )
      Contact( #Trig_Vill )
      Contact( #power_Vill )
      wire#w6
      Coil( "HS".Forks_Pitcher.OnCom )
      P_Trig( #ramp_sync_old )
      Coil( "ALG".RampSyncSig )
   END_RUNG
   RUNG wire#w2
      Contact( #ForksForcingFinish )
   END_RUNG wire#w3
   RUNG wire#w4
      Contact( "S16.2" )
      { S7_Templates := "SrcType := Int" } EQ_Contact(in1 := #LayersCounter, in2 := 0)
   END_RUNG wire#w5
   RUNG wire#w6
      Contact( "B15.7" )
      S_ODT(T_NO := "Tag_19(1)", TV := s5t#1s, R :=, BI =>, RET_VAL =>)
      Coil( "IM_PFM".M_233_Fork_PFM.OnCom )
   END_RUNG
   RUNG wire#w5
      Not()
      Contact( "Tag_34" )
      Coil( #AlarmLowerElevator )
      Contact( #NoGasketMode )
      S_Coil( #ElevatorLowering )
   END_RUNG
   RUNG wire#w1
      Contact( #Trig_Vill2 )
      wire#w7
      Coil( "HS".Forks_Pitcher.OffCom )
   END_RUNG
   RUNG wire#w7
      Contact( "B15.5" )
      S_ODT(T_NO := "M213AlarmFilter", TV := s5t#1s, R :=, BI =>, RET_VAL =>)
      Coil( "IM_PFM".M_233_Fork_PFM.OffCom )
   END_RUNG
   // the same network as SCL:
   #_w1 := NOT "ALG".Alarm_Sorting AND "ALG".Auto_Sorting;
   "Tag_34" := #_w1 AND #HaveSxema AND (("ServDB".QPlanksInLayer = #BoardInLayerCounter) OR #ForksForcingFinish);
   #_w2 := "Tag_34" AND "Tag_46" AND ((NOT "FC_232_1" AND NOT "FC_232_2") OR ("S16.2" AND (#LayersCounter = 0)));
   "HS".Forks_Pitcher.OnCom := #_w2 AND #Trig_Dovod AND NOT #LiftPushingPacket AND NOT "S18.3" AND #RampIsOn AND #Trig_Vill AND #power_Vill;
   #_w3 := "HS".Forks_Pitcher.OnCom AND NOT #ramp_sync_old;   // rising edge
   #ramp_sync_old := "HS".Forks_Pitcher.OnCom;
   "ALG".RampSyncSig := #_w3;
   #_s5time1 := S_ODT(T_NO := "Tag_19(1)", S := "HS".Forks_Pitcher.OnCom AND "B15.7", TV := s5t#1s, Q => #_w4);
   "IM_PFM".M_233_Fork_PFM.OnCom := #_w4;
   #AlarmLowerElevator := NOT #_w2 AND "Tag_34";
   IF #AlarmLowerElevator AND #NoGasketMode THEN #ElevatorLowering := TRUE; END_IF;
   "HS".Forks_Pitcher.OffCom := #_w1 AND #Trig_Vill2;
   #_s5time2 := S_ODT(T_NO := "M213AlarmFilter",
                      S := "HS".Forks_Pitcher.OffCom AND "B15.5",
                      TV := s5t#1s,
                      Q => #_w5);
   "IM_PFM".M_233_Fork_PFM.OffCom := #_w5;
END_REGION

REGION Network 41: Скорость вил ПЧТ
   RUNG wire#powerrail
      UNSCALE(IN := "IM_PFM".M_233_Fork_PFM.SetSpeed, HI_LIM := 50.0, LO_LIM := -50.0, BIPOLAR := "TRUE", RET_VAL => #Sert, OUT => "K1-233U":P)
   END_RUNG
   // the same network as SCL:
   #Sert := UNSCALE(IN := "IM_PFM".M_233_Fork_PFM.SetSpeed,
                    HI_LIM := 50.0,
                    LO_LIM := -50.0,
                    BIPOLAR := "TRUE",
                    OUT => "K1-233U":P);
END_REGION

REGION Network 42: триггер доводчика
   RUNG wire#powerrail
      Contact( "Tag_34" )
      Contact( "B18.6" )
      S_ODT(T_NO := "Tag_76", TV := s5t#2500ms, R :=, BI =>, RET_VAL =>)
      S_SR(operand := #Trig_Dovod, r1 := wire#w1)
   END_RUNG
   RUNG wire#powerrail
      Contact( "S15.2" )
   END_RUNG wire#w1
   RUNG wire#powerrail
      Contact( "S76.2" )
   END_RUNG wire#w1
   // the same network as SCL:
   #_s5time1 := S_ODT(T_NO := "Tag_76", S := "Tag_34" AND "B18.6", TV := s5t#2500ms, Q => #_w1);
   IF #_w1 THEN
       #Trig_Dovod := TRUE;   // SR flip-flop
   END_IF;
   IF "S15.2" OR "S76.2" THEN #Trig_Dovod := FALSE; END_IF;
END_REGION

REGION Network 43: задержка на доводчик
   // no SCL statement known for SfCoil: written as a call
   SfCoil(in := "B14.4" OR "B14.5", value := s5t#50ms, operand := "DelayDovodPFM");
END_REGION

REGION Network 44: M 325 авто вперед
   RUNG wire#powerrail
      I_Contact( "ALG".Alarm_Sorting )
      Contact( "ALG".Auto_Sorting )
      wire#w1
      Contact( "Tag_34" )
      I_Contact( #Trig_Dovod )
      wire#w2
      I_Contact( "UporPFM_DB".CommonAlarm )
      I_Contact( "SensLineAlarms" )
      Coil( "IM".M_325_Tr_Hill.OnCom )
   END_RUNG
   RUNG wire#w1
      Contact( "DelayDovodPFM" )
   END_RUNG wire#w2
   // the same network as SCL:
   "IM".M_325_Tr_Hill.OnCom := NOT "ALG".Alarm_Sorting AND "ALG".Auto_Sorting AND (("Tag_34" AND NOT #Trig_Dovod) OR "DelayDovodPFM") AND NOT "UporPFM_DB".CommonAlarm AND NOT "SensLineAlarms";
END_REGION

REGION Network 45: Старт ПЧТ 325
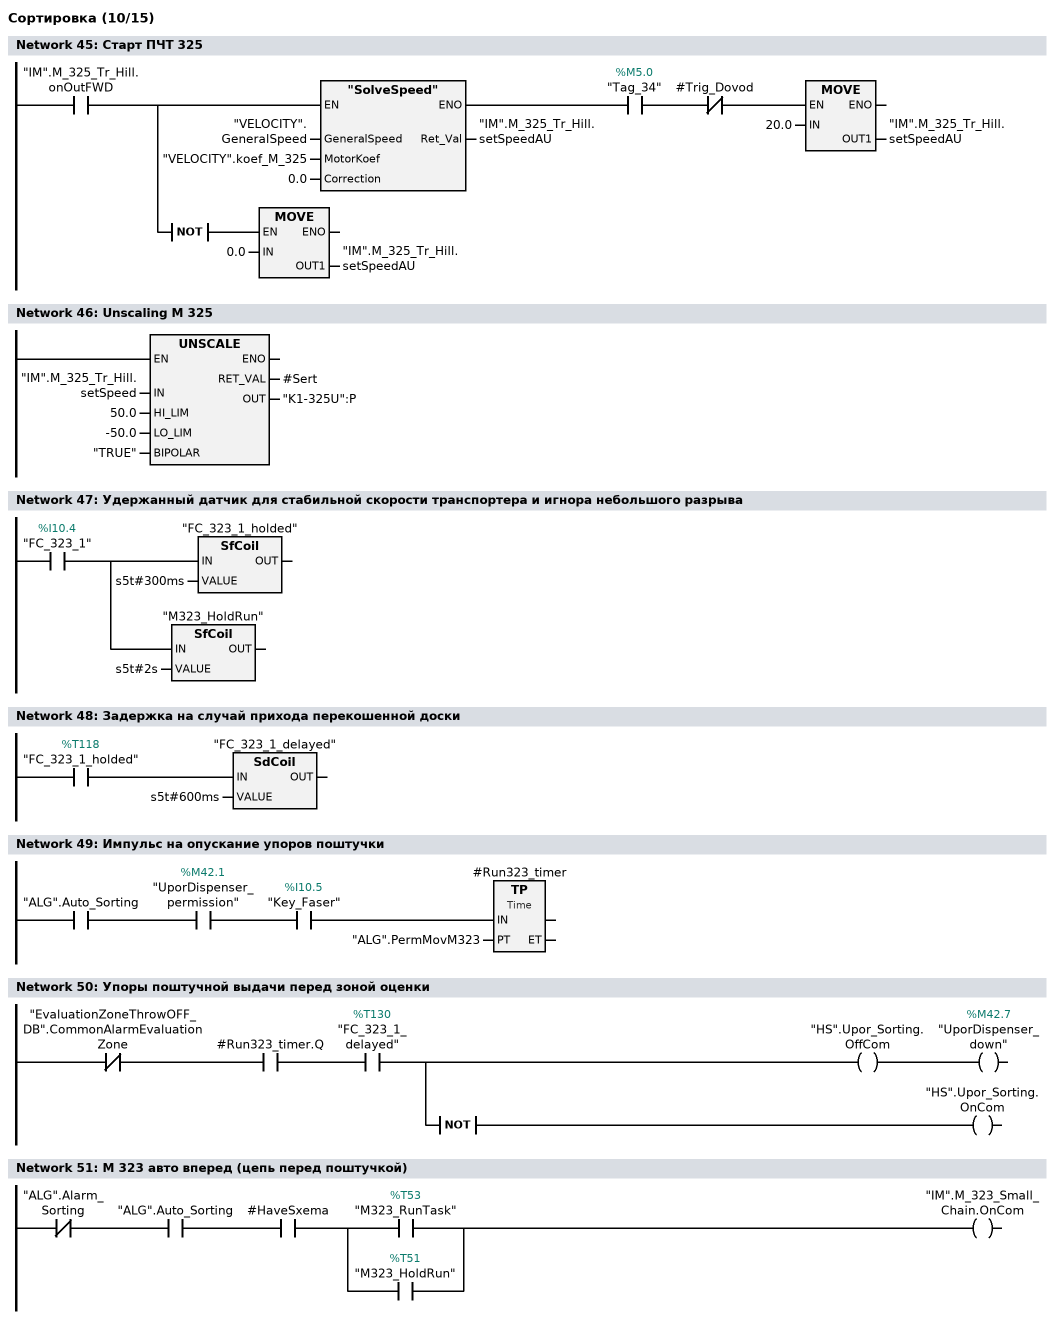
   RUNG wire#powerrail
      Contact( "IM".M_325_Tr_Hill.onOutFWD )
      wire#w1
      "SolveSpeed"(GeneralSpeed := "VELOCITY".GeneralSpeed, MotorKoef := "VELOCITY".koef_M_325, Correction := 0.0, Ret_Val => "IM".M_325_Tr_Hill.setSpeedAU)
      Contact( "Tag_34" )
      I_Contact( #Trig_Dovod )
      { S7_GenerateENO := "TRUE" } Move(in := 20.0, out1 => "IM".M_325_Tr_Hill.setSpeedAU)
   END_RUNG
   RUNG wire#w1
      Not()
      { S7_GenerateENO := "TRUE" } Move(in := 0.0, out1 => "IM".M_325_Tr_Hill.setSpeedAU)
   END_RUNG
   // the same network as SCL:
   #_w2 := "IM".M_325_Tr_Hill.onOutFWD;
   "IM".M_325_Tr_Hill.setSpeedAU := "SolveSpeed"(EN := "IM".M_325_Tr_Hill.onOutFWD,
                           GeneralSpeed := "VELOCITY".GeneralSpeed,
                           MotorKoef := "VELOCITY".koef_M_325,
                           Correction := 0.0,
                           ENO => #_w1);
   IF #_w1 AND "Tag_34" AND NOT #Trig_Dovod THEN "IM".M_325_Tr_Hill.setSpeedAU := 20.0; END_IF;
   IF NOT #_w2 THEN "IM".M_325_Tr_Hill.setSpeedAU := 0.0; END_IF;
END_REGION

REGION Network 46: Unscaling M 325
   RUNG wire#powerrail
      UNSCALE(IN := "IM".M_325_Tr_Hill.setSpeed, HI_LIM := 50.0, LO_LIM := -50.0, BIPOLAR := "TRUE", RET_VAL => #Sert, OUT => "K1-325U":P)
   END_RUNG
   // the same network as SCL:
   #Sert := UNSCALE(IN := "IM".M_325_Tr_Hill.setSpeed,
                    HI_LIM := 50.0,
                    LO_LIM := -50.0,
                    BIPOLAR := "TRUE",
                    OUT => "K1-325U":P);
END_REGION

REGION Network 47: Удержанный датчик для стабильной скорости транспортера и игнора небольшого разрыва
   // no SCL statement known for SfCoil: written as a call
   #_w1 := "FC_323_1";
   SfCoil(in := "FC_323_1", value := s5t#300ms, operand := "FC_323_1_holded");
   SfCoil(in := #_w1, value := s5t#2s, operand := "M323_HoldRun");
END_REGION

REGION Network 48: Задержка на случай прихода перекошенной доски
   // no SCL statement known for SdCoil: written as a call
   SdCoil(in := "FC_323_1_holded", value := s5t#600ms, operand := "FC_323_1_delayed");
END_REGION

REGION Network 49: Импульс на опускание упоров поштучки
   RUNG wire#powerrail
      Contact( "ALG".Auto_Sorting )
      Contact( "UporDispenser_permission" )
      Contact( "Key_Faser" )
      { S7_Templates := "time_type := Time" } #Run323_timer.TP(pt := "ALG".PermMovM323, et =>)
   END_RUNG
   // the same network as SCL:
   #Run323_timer.TP(IN := "ALG".Auto_Sorting AND "UporDispenser_permission" AND "Key_Faser",
                    PT := "ALG".PermMovM323);
END_REGION

REGION Network 50: Упоры поштучной выдачи перед зоной оценки
   RUNG wire#powerrail
      I_Contact( "EvaluationZoneThrowOFF_DB".CommonAlarmEvaluationZone )
      Contact( #Run323_timer.Q )
      Contact( "FC_323_1_delayed" )
      wire#w1
      Coil( "HS".Upor_Sorting.OffCom )
      Coil( "UporDispenser_down" )
   END_RUNG
   RUNG wire#w1
      Not()
      Coil( "HS".Upor_Sorting.OnCom )
   END_RUNG
   // the same network as SCL:
   "HS".Upor_Sorting.OffCom := NOT "EvaluationZoneThrowOFF_DB".CommonAlarmEvaluationZone AND #Run323_timer.Q AND "FC_323_1_delayed";
   "UporDispenser_down" := "HS".Upor_Sorting.OffCom;
   "HS".Upor_Sorting.OnCom := NOT "HS".Upor_Sorting.OffCom;
END_REGION

REGION Network 51: M 323 авто вперед (цепь перед поштучкой)
   RUNG wire#powerrail
      I_Contact( "ALG".Alarm_Sorting )
      Contact( "ALG".Auto_Sorting )
      Contact( #HaveSxema )
      wire#w1
      Contact( "M323_RunTask" )
      wire#w2
      Coil( "IM".M_323_Small_Chain.OnCom )
   END_RUNG
   RUNG wire#w1
      Contact( "M323_HoldRun" )
   END_RUNG wire#w2
   // the same network as SCL:
   "IM".M_323_Small_Chain.OnCom := NOT "ALG".Alarm_Sorting AND "ALG".Auto_Sorting AND #HaveSxema AND ("M323_RunTask" OR "M323_HoldRun");
END_REGION

REGION Network 52: Старт ПЧТ M 323
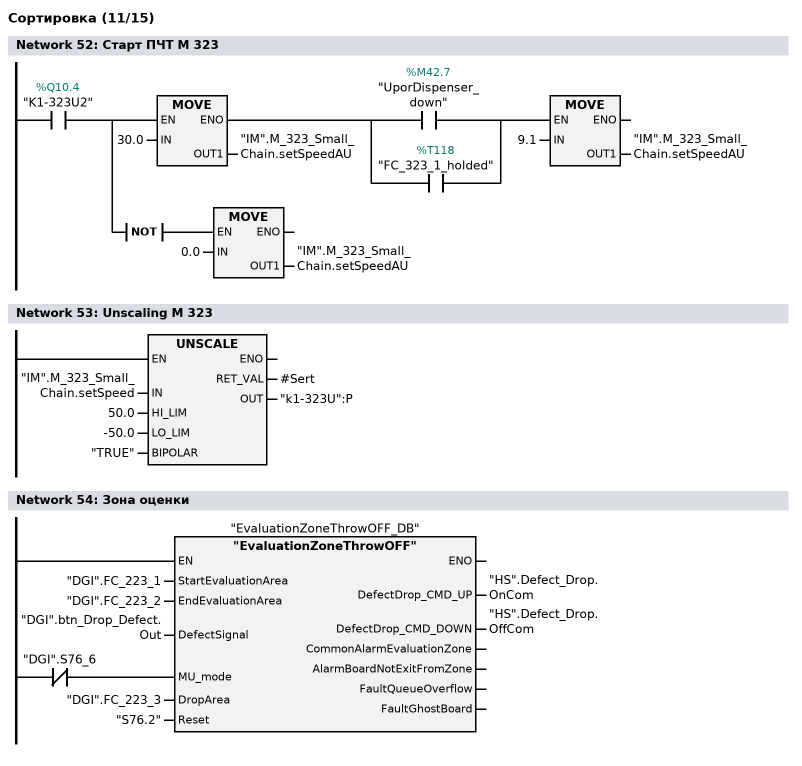
   RUNG wire#powerrail
      Contact( "K1-323U2" )
      wire#w1
      { S7_GenerateENO := "TRUE" } Move(in := 30.0, out1 => "IM".M_323_Small_Chain.setSpeedAU)
      wire#w2
      Contact( "UporDispenser_down" )
      wire#w3
      { S7_GenerateENO := "TRUE" } Move(in := 9.1, out1 => "IM".M_323_Small_Chain.setSpeedAU)
   END_RUNG
   RUNG wire#w2
      Contact( "FC_323_1_holded" )
   END_RUNG wire#w3
   RUNG wire#w1
      Not()
      { S7_GenerateENO := "TRUE" } Move(in := 0.0, out1 => "IM".M_323_Small_Chain.setSpeedAU)
   END_RUNG
   // the same network as SCL:
   // ENO of a box is taken as its EN; it also drops when the box reports an error
   IF "K1-323U2" THEN "IM".M_323_Small_Chain.setSpeedAU := 30.0; END_IF;
   IF "K1-323U2" AND ("UporDispenser_down" OR "FC_323_1_holded") THEN
       "IM".M_323_Small_Chain.setSpeedAU := 9.1;
   END_IF;
   IF NOT "K1-323U2" THEN "IM".M_323_Small_Chain.setSpeedAU := 0.0; END_IF;
END_REGION

REGION Network 53: Unscaling M 323
   RUNG wire#powerrail
      UNSCALE(IN := "IM".M_323_Small_Chain.setSpeed, HI_LIM := 50.0, LO_LIM := -50.0, BIPOLAR := "TRUE", RET_VAL => #Sert, OUT => "k1-323U":P)
   END_RUNG
   // the same network as SCL:
   #Sert := UNSCALE(IN := "IM".M_323_Small_Chain.setSpeed,
                    HI_LIM := 50.0,
                    LO_LIM := -50.0,
                    BIPOLAR := "TRUE",
                    OUT => "k1-323U":P);
END_REGION

REGION Network 54: Зона оценки
   RUNG wire#powerrail
      "EvaluationZoneThrowOFF_DB"(MU_mode := wire#w1, StartEvaluationArea := "DGI".FC_223_1, EndEvaluationArea := "DGI".FC_223_2, DefectSignal := "DGI".btn_Drop_Defect.Out, DropArea := "DGI".FC_223_3, Reset := "S76.2", DefectDrop_CMD_UP => "HS".Defect_Drop.OnCom, DefectDrop_CMD_DOWN => "HS".Defect_Drop.OffCom, CommonAlarmEvaluationZone =>, AlarmBoardNotExitFromZone =>, FaultQueueOverflow =>, FaultGhostBoard =>)
   END_RUNG
   RUNG wire#powerrail
      I_Contact( "DGI".S76_6 )
   END_RUNG wire#w1
   // the same network as SCL:
   "EvaluationZoneThrowOFF_DB"(StartEvaluationArea := "DGI".FC_223_1,   // "EvaluationZoneThrowOFF"
                           EndEvaluationArea := "DGI".FC_223_2,
                           DefectSignal := "DGI".btn_Drop_Defect.Out,
                           MU_mode := NOT "DGI".S76_6,
                           DropArea := "DGI".FC_223_3,
                           Reset := "S76.2",
                           DefectDrop_CMD_UP => "HS".Defect_Drop.OnCom,
                           DefectDrop_CMD_DOWN => "HS".Defect_Drop.OffCom);
END_REGION

REGION Network 55: Измерение длины досок + залипание линейки + управление очередью бобышек под линейкой
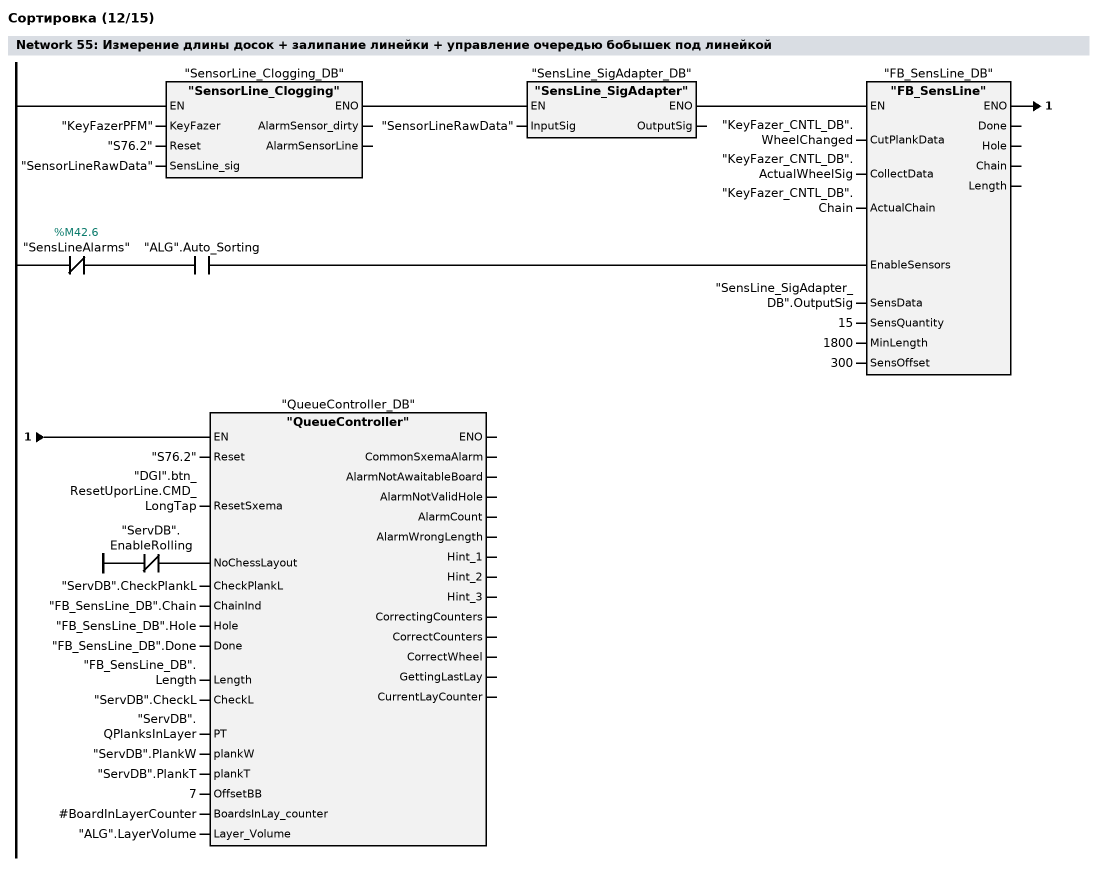
   RUNG wire#powerrail
      "SensorLine_Clogging_DB"(KeyFazer := "KeyFazerPFM", Reset := "S76.2", SensLine_sig := "SensorLineRawData", AlarmSensor_dirty =>, AlarmSensorLine =>)
      "SensLine_SigAdapter_DB"(InputSig := "SensorLineRawData", OutputSig =>)
      "FB_SensLine_DB"(EnableSensors := wire#w1, CutPlankData := "KeyFazer_CNTL_DB".WheelChanged, CollectData := "KeyFazer_CNTL_DB".ActualWheelSig, ActualChain := "KeyFazer_CNTL_DB".Chain, SensData := "SensLine_SigAdapter_DB".OutputSig, SensQuantity := 15, MinLength := 1800, SensOffset := 300, Done =>, Hole =>, Chain =>, Length =>)
      "QueueController_DB"(NoChessLayout := wire#w2, Reset := "S76.2", ResetSxema := "DGI".btn_ResetUporLine.CMD_LongTap, CheckPlankL := "ServDB".CheckPlankL, ChainInd := "FB_SensLine_DB".Chain, Hole := "FB_SensLine_DB".Hole, Done := "FB_SensLine_DB".Done, Length := "FB_SensLine_DB".Length, CheckL := "ServDB".CheckL, PT := "ServDB".QPlanksInLayer, plankW := "ServDB".PlankW, plankT := "ServDB".PlankT, OffsetBB := 7, BoardsInLay_counter := #BoardInLayerCounter, Layer_Volume := "ALG".LayerVolume, CommonSxemaAlarm =>, AlarmNotAwaitableBoard =>, AlarmNotValidHole =>, AlarmCount =>, AlarmWrongLength =>, Hint_1 =>, Hint_2 =>, Hint_3 =>, CorrectingCounters =>, CorrectCounters =>, CorrectWheel =>, GettingLastLay =>, CurrentLayCounter =>)
   END_RUNG
   RUNG wire#powerrail
      I_Contact( "SensLineAlarms" )
      Contact( "ALG".Auto_Sorting )
   END_RUNG wire#w1
   RUNG wire#powerrail
      I_Contact( "ServDB".EnableRolling )
   END_RUNG wire#w2
   // the same network as SCL:
   "SensorLine_Clogging_DB"(KeyFazer := "KeyFazerPFM",   // "SensorLine_Clogging"
                           Reset := "S76.2",
                           SensLine_sig := "SensorLineRawData",
                           ENO => #_w1);
   "SensLine_SigAdapter_DB"(EN := #_w1, InputSig := "SensorLineRawData", ENO => #_w2);   // "SensLine_SigAdapter"
   "FB_SensLine_DB"(EN := #_w2,   // "FB_SensLine"
                    CutPlankData := "KeyFazer_CNTL_DB".WheelChanged,
                    CollectData := "KeyFazer_CNTL_DB".ActualWheelSig,
                    ActualChain := "KeyFazer_CNTL_DB".Chain,
                    EnableSensors := NOT "SensLineAlarms" AND "ALG".Auto_Sorting,
                    SensData := "SensLine_SigAdapter_DB".OutputSig,
                    SensQuantity := 15,
                    MinLength := 1800,
                    SensOffset := 300,
                    ENO => #_w3);
   IF #_w3 THEN
       "QueueController_DB"(Reset := "S76.2",   // "QueueController"
                            ResetSxema := "DGI".btn_ResetUporLine.CMD_LongTap,
                            NoChessLayout := NOT "ServDB".EnableRolling,
                            CheckPlankL := "ServDB".CheckPlankL,
                            ChainInd := "FB_SensLine_DB".Chain,
                            Hole := "FB_SensLine_DB".Hole,
                            Done := "FB_SensLine_DB".Done,
                            Length := "FB_SensLine_DB".Length,
                            CheckL := "ServDB".CheckL,
                            PT := "ServDB".QPlanksInLayer,
                            plankW := "ServDB".PlankW,
                            plankT := "ServDB".PlankT,
                            OffsetBB := 7,
                            BoardsInLay_counter := #BoardInLayerCounter,
                            Layer_Volume := "ALG".LayerVolume);
   END_IF;
END_REGION

REGION Network 56: Управление упорами перед транспортером с бобышками
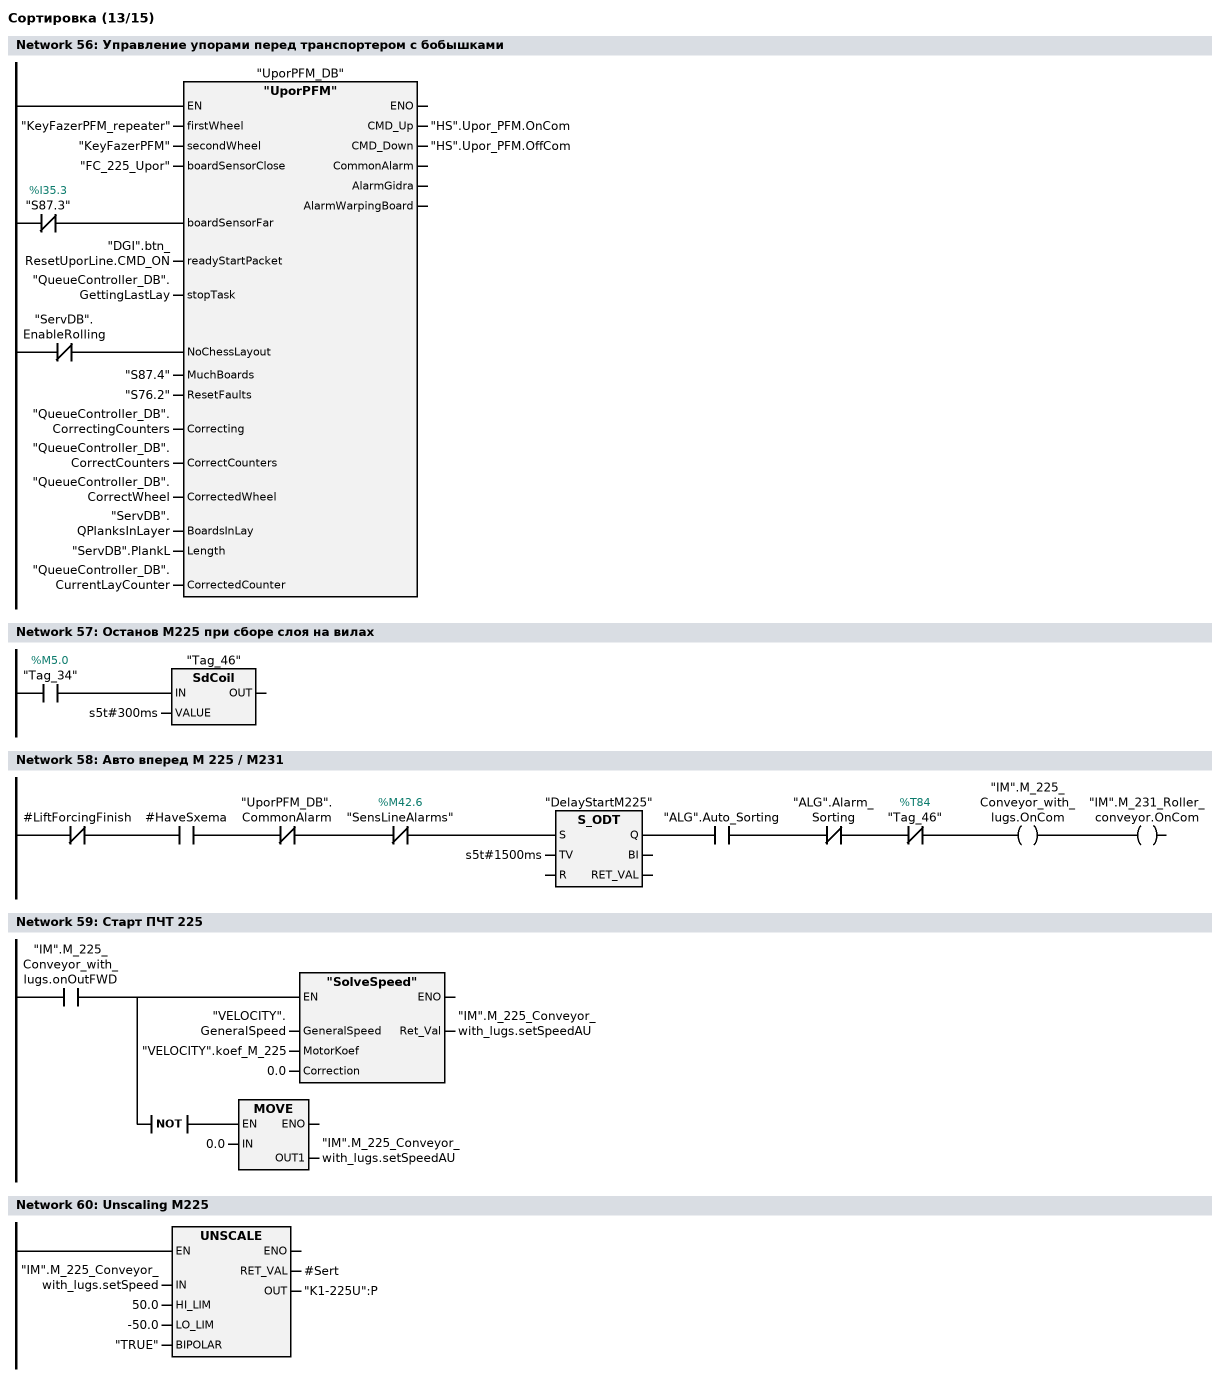
   RUNG wire#powerrail
      "UporPFM_DB"(boardSensorFar := wire#w1, NoChessLayout := wire#w2, firstWheel := "KeyFazerPFM_repeater", secondWheel := "KeyFazerPFM", boardSensorClose := "FC_225_Upor", readyStartPacket := "DGI".btn_ResetUporLine.CMD_ON, stopTask := "QueueController_DB".GettingLastLay, MuchBoards := "S87.4", ResetFaults := "S76.2", Correcting := "QueueController_DB".CorrectingCounters, CorrectCounters := "QueueController_DB".CorrectCounters, CorrectedWheel := "QueueController_DB".CorrectWheel, BoardsInLay := "ServDB".QPlanksInLayer, Length := "ServDB".PlankL, CorrectedCounter := "QueueController_DB".CurrentLayCounter, CMD_Up => "HS".Upor_PFM.OnCom, CMD_Down => "HS".Upor_PFM.OffCom, CommonAlarm =>, AlarmGidra =>, AlarmWarpingBoard =>)
   END_RUNG
   RUNG wire#powerrail
      I_Contact( "S87.3" )
   END_RUNG wire#w1
   RUNG wire#powerrail
      I_Contact( "ServDB".EnableRolling )
   END_RUNG wire#w2
   // the same network as SCL:
   "UporPFM_DB"(firstWheel := "KeyFazerPFM_repeater",   // "UporPFM"
                secondWheel := "KeyFazerPFM",
                boardSensorClose := "FC_225_Upor",
                boardSensorFar := NOT "S87.3",
                readyStartPacket := "DGI".btn_ResetUporLine.CMD_ON,
                stopTask := "QueueController_DB".GettingLastLay,
                NoChessLayout := NOT "ServDB".EnableRolling,
                MuchBoards := "S87.4",
                ResetFaults := "S76.2",
                Correcting := "QueueController_DB".CorrectingCounters,
                CorrectCounters := "QueueController_DB".CorrectCounters,
                CorrectedWheel := "QueueController_DB".CorrectWheel,
                BoardsInLay := "ServDB".QPlanksInLayer,
                Length := "ServDB".PlankL,
                CorrectedCounter := "QueueController_DB".CurrentLayCounter,
                CMD_Up => "HS".Upor_PFM.OnCom,
                CMD_Down => "HS".Upor_PFM.OffCom);
END_REGION

REGION Network 57: Останов M225 при сборе слоя на вилах
   // no SCL statement known for SdCoil: written as a call
   SdCoil(in := "Tag_34", value := s5t#300ms, operand := "Tag_46");
END_REGION

REGION Network 58: Авто вперед M 225 / M231
   RUNG wire#powerrail
      I_Contact( #LiftForcingFinish )
      Contact( #HaveSxema )
      I_Contact( "UporPFM_DB".CommonAlarm )
      I_Contact( "SensLineAlarms" )
      S_ODT(T_NO := "DelayStartM225", TV := s5t#1500ms, R :=, BI =>, RET_VAL =>)
      Contact( "ALG".Auto_Sorting )
      I_Contact( "ALG".Alarm_Sorting )
      I_Contact( "Tag_46" )
      Coil( "IM".M_225_Conveyor_with_lugs.OnCom )
      Coil( "IM".M_231_Roller_conveyor.OnCom )
   END_RUNG
   // the same network as SCL:
   #_s5time1 := S_ODT(T_NO := "DelayStartM225",
                      S := NOT #LiftForcingFinish AND #HaveSxema AND NOT "UporPFM_DB".CommonAlarm AND NOT "SensLineAlarms",
                      TV := s5t#1500ms,
                      Q => #_w1);
   "IM".M_225_Conveyor_with_lugs.OnCom := #_w1 AND "ALG".Auto_Sorting AND NOT "ALG".Alarm_Sorting AND NOT "Tag_46";
   "IM".M_231_Roller_conveyor.OnCom := "IM".M_225_Conveyor_with_lugs.OnCom;
END_REGION

REGION Network 59: Старт ПЧТ 225
   RUNG wire#powerrail
      Contact( "IM".M_225_Conveyor_with_lugs.onOutFWD )
      wire#w1
      "SolveSpeed"(GeneralSpeed := "VELOCITY".GeneralSpeed, MotorKoef := "VELOCITY".koef_M_225, Correction := 0.0, Ret_Val => "IM".M_225_Conveyor_with_lugs.setSpeedAU)
   END_RUNG
   RUNG wire#w1
      Not()
      { S7_GenerateENO := "TRUE" } Move(in := 0.0, out1 => "IM".M_225_Conveyor_with_lugs.setSpeedAU)
   END_RUNG
   // the same network as SCL:
   #_w1 := "IM".M_225_Conveyor_with_lugs.onOutFWD;
   IF #_w1 THEN
       "IM".M_225_Conveyor_with_lugs.setSpeedAU := "SolveSpeed"(GeneralSpeed := "VELOCITY".GeneralSpeed,
                               MotorKoef := "VELOCITY".koef_M_225,
                               Correction := 0.0);
   END_IF;
   IF NOT #_w1 THEN "IM".M_225_Conveyor_with_lugs.setSpeedAU := 0.0; END_IF;
END_REGION

REGION Network 60: Unscaling M225
   RUNG wire#powerrail
      UNSCALE(IN := "IM".M_225_Conveyor_with_lugs.setSpeed, HI_LIM := 50.0, LO_LIM := -50.0, BIPOLAR := "TRUE", RET_VAL => #Sert, OUT => "K1-225U":P)
   END_RUNG
   // the same network as SCL:
   #Sert := UNSCALE(IN := "IM".M_225_Conveyor_with_lugs.setSpeed,
                    HI_LIM := 50.0,
                    LO_LIM := -50.0,
                    BIPOLAR := "TRUE",
                    OUT => "K1-225U":P);
END_REGION

REGION Network 61: Старт ПЧТ 231
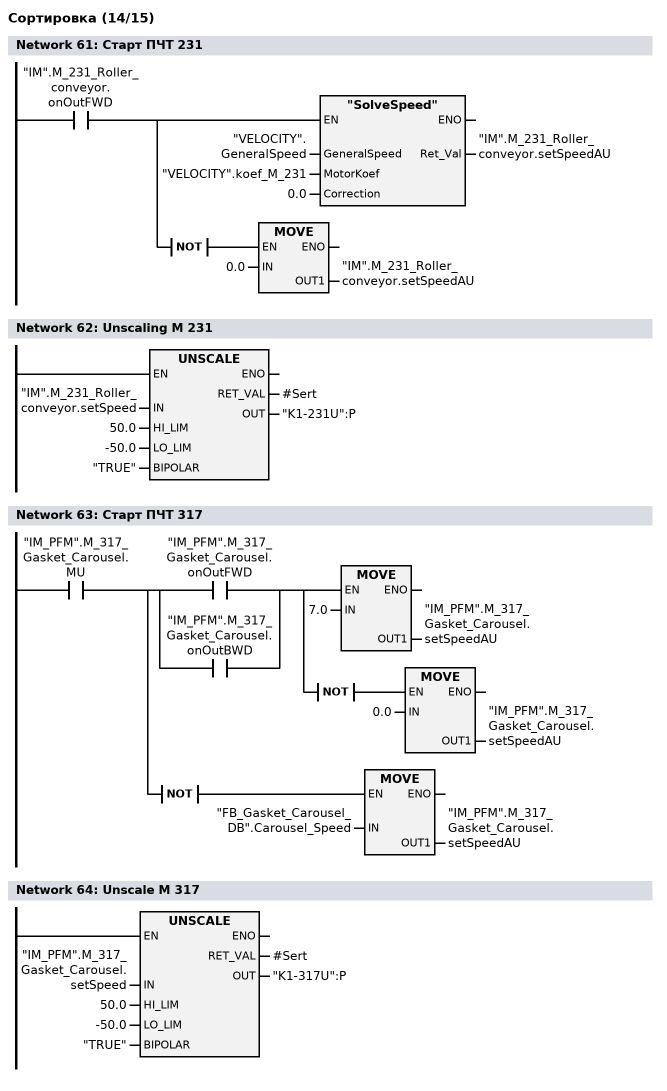
   RUNG wire#powerrail
      Contact( "IM".M_231_Roller_conveyor.onOutFWD )
      wire#w1
      "SolveSpeed"(GeneralSpeed := "VELOCITY".GeneralSpeed, MotorKoef := "VELOCITY".koef_M_231, Correction := 0.0, Ret_Val => "IM".M_231_Roller_conveyor.setSpeedAU)
   END_RUNG
   RUNG wire#w1
      Not()
      { S7_GenerateENO := "TRUE" } Move(in := 0.0, out1 => "IM".M_231_Roller_conveyor.setSpeedAU)
   END_RUNG
   // the same network as SCL:
   #_w1 := "IM".M_231_Roller_conveyor.onOutFWD;
   IF #_w1 THEN
       "IM".M_231_Roller_conveyor.setSpeedAU := "SolveSpeed"(GeneralSpeed := "VELOCITY".GeneralSpeed,
                               MotorKoef := "VELOCITY".koef_M_231,
                               Correction := 0.0);
   END_IF;
   IF NOT #_w1 THEN "IM".M_231_Roller_conveyor.setSpeedAU := 0.0; END_IF;
END_REGION

REGION Network 62: Unscaling M 231
   RUNG wire#powerrail
      UNSCALE(IN := "IM".M_231_Roller_conveyor.setSpeed, HI_LIM := 50.0, LO_LIM := -50.0, BIPOLAR := "TRUE", RET_VAL => #Sert, OUT => "K1-231U":P)
   END_RUNG
   // the same network as SCL:
   #Sert := UNSCALE(IN := "IM".M_231_Roller_conveyor.setSpeed,
                    HI_LIM := 50.0,
                    LO_LIM := -50.0,
                    BIPOLAR := "TRUE",
                    OUT => "K1-231U":P);
END_REGION

REGION Network 63: Старт ПЧТ 317
   RUNG wire#powerrail
      Contact( "IM_PFM".M_317_Gasket_Carousel.MU )
      wire#w1
      Contact( "IM_PFM".M_317_Gasket_Carousel.onOutFWD )
      wire#w2
      { S7_GenerateENO := "TRUE" } Move(in := 7.0, out1 => "IM_PFM".M_317_Gasket_Carousel.setSpeedAU)
   END_RUNG
   RUNG wire#w1
      Contact( "IM_PFM".M_317_Gasket_Carousel.onOutBWD )
   END_RUNG wire#w2
   RUNG wire#w2
      Not()
      { S7_GenerateENO := "TRUE" } Move(in := 0.0, out1 => "IM_PFM".M_317_Gasket_Carousel.setSpeedAU)
   END_RUNG
   RUNG wire#w1
      Not()
      { S7_GenerateENO := "TRUE" } Move(in := "FB_Gasket_Carousel_DB".Carousel_Speed, out1 => "IM_PFM".M_317_Gasket_Carousel.setSpeedAU)
   END_RUNG
   // the same network as SCL:
   #_w1 := "IM_PFM".M_317_Gasket_Carousel.MU AND ("IM_PFM".M_317_Gasket_Carousel.onOutFWD OR "IM_PFM".M_317_Gasket_Carousel.onOutBWD);
   IF #_w1 THEN "IM_PFM".M_317_Gasket_Carousel.setSpeedAU := 7.0; END_IF;
   IF NOT #_w1 THEN "IM_PFM".M_317_Gasket_Carousel.setSpeedAU := 0.0; END_IF;
   IF NOT "IM_PFM".M_317_Gasket_Carousel.MU THEN
       "IM_PFM".M_317_Gasket_Carousel.setSpeedAU := "FB_Gasket_Carousel_DB".Carousel_Speed;
   END_IF;
END_REGION

REGION Network 64: Unscale M 317
   RUNG wire#powerrail
      UNSCALE(IN := "IM_PFM".M_317_Gasket_Carousel.setSpeed, HI_LIM := 50.0, LO_LIM := -50.0, BIPOLAR := "TRUE", RET_VAL => #Sert, OUT => "K1-317U":P)
   END_RUNG
   // the same network as SCL:
   #Sert := UNSCALE(IN := "IM_PFM".M_317_Gasket_Carousel.setSpeed,
                    HI_LIM := 50.0,
                    LO_LIM := -50.0,
                    BIPOLAR := "TRUE",
                    OUT => "K1-317U":P);
END_REGION

REGION Network 65: Логика рамы прокладок
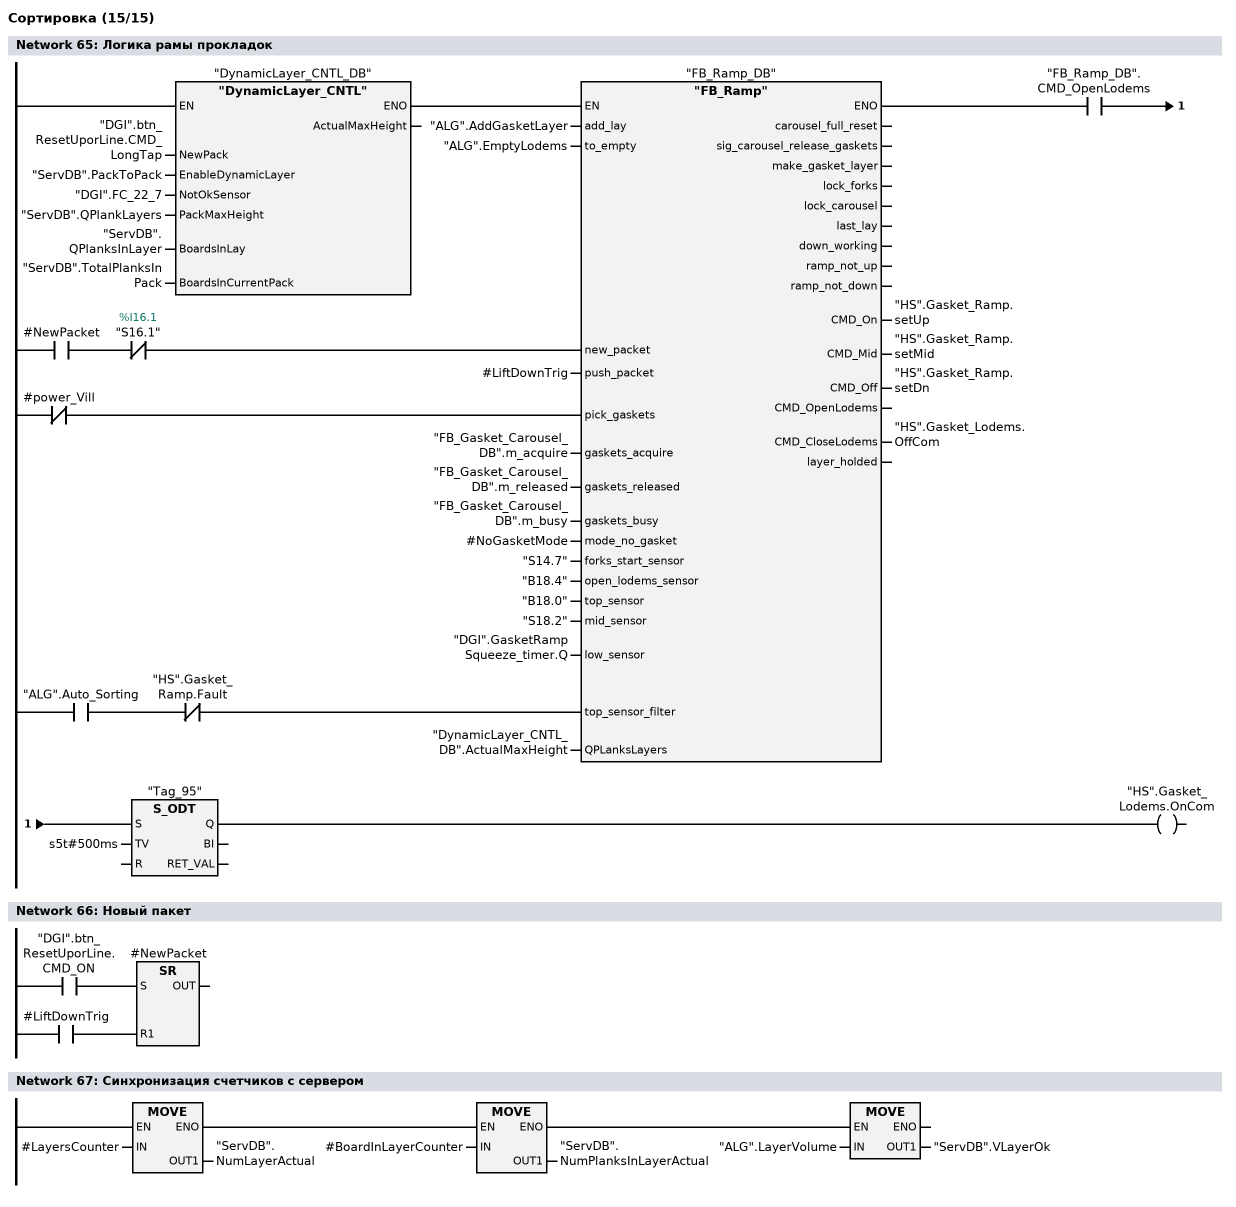
   RUNG wire#powerrail
      "DynamicLayer_CNTL_DB"(NewPack := "DGI".btn_ResetUporLine.CMD_LongTap, EnableDynamicLayer := "ServDB".PackToPack, NotOkSensor := "DGI".FC_22_7, PackMaxHeight := "ServDB".QPlankLayers, BoardsInLay := "ServDB".QPlanksInLayer, BoardsInCurrentPack := "ServDB".TotalPlanksInPack, ActualMaxHeight =>)
      "FB_Ramp_DB"(new_packet := wire#w1, pick_gaskets := wire#w2, top_sensor_filter := wire#w3, add_lay := "ALG".AddGasketLayer, to_empty := "ALG".EmptyLodems, push_packet := #LiftDownTrig, gaskets_acquire := "FB_Gasket_Carousel_DB".m_acquire, gaskets_released := "FB_Gasket_Carousel_DB".m_released, gaskets_busy := "FB_Gasket_Carousel_DB".m_busy, mode_no_gasket := #NoGasketMode, forks_start_sensor := "S14.7", open_lodems_sensor := "B18.4", top_sensor := "B18.0", mid_sensor := "S18.2", low_sensor := "DGI".GasketRampSqueeze_timer.Q, QPLanksLayers := "DynamicLayer_CNTL_DB".ActualMaxHeight, carousel_full_reset =>, sig_carousel_release_gaskets =>, make_gasket_layer =>, lock_forks =>, lock_carousel =>, last_lay =>, down_working =>, ramp_not_up =>, ramp_not_down =>, CMD_On => "HS".Gasket_Ramp.setUp, CMD_Mid => "HS".Gasket_Ramp.setMid, CMD_Off => "HS".Gasket_Ramp.setDn, CMD_OpenLodems =>, CMD_CloseLodems => "HS".Gasket_Lodems.OffCom, layer_holded =>)
      Contact( "FB_Ramp_DB".CMD_OpenLodems )
      S_ODT(T_NO := "Tag_95", TV := s5t#500ms, R :=, BI =>, RET_VAL =>)
      Coil( "HS".Gasket_Lodems.OnCom )
   END_RUNG
   RUNG wire#powerrail
      Contact( #NewPacket )
      I_Contact( "S16.1" )
   END_RUNG wire#w1
   RUNG wire#powerrail
      I_Contact( #power_Vill )
   END_RUNG wire#w2
   RUNG wire#powerrail
      Contact( "ALG".Auto_Sorting )
      I_Contact( "HS".Gasket_Ramp.Fault )
   END_RUNG wire#w3
   // the same network as SCL:
   "DynamicLayer_CNTL_DB"(NewPack := "DGI".btn_ResetUporLine.CMD_LongTap,   // "DynamicLayer_CNTL"
                          EnableDynamicLayer := "ServDB".PackToPack,
                          NotOkSensor := "DGI".FC_22_7,
                          PackMaxHeight := "ServDB".QPlankLayers,
                          BoardsInLay := "ServDB".QPlanksInLayer,
                          BoardsInCurrentPack := "ServDB".TotalPlanksInPack,
                          ENO => #_w1);
   "FB_Ramp_DB"(EN := #_w1,   // "FB_Ramp"
                add_lay := "ALG".AddGasketLayer,
                to_empty := "ALG".EmptyLodems,
                new_packet := #NewPacket AND NOT "S16.1",
                push_packet := #LiftDownTrig,
                pick_gaskets := NOT #power_Vill,
                gaskets_acquire := "FB_Gasket_Carousel_DB".m_acquire,
                gaskets_released := "FB_Gasket_Carousel_DB".m_released,
                gaskets_busy := "FB_Gasket_Carousel_DB".m_busy,
                mode_no_gasket := #NoGasketMode,
                forks_start_sensor := "S14.7",
                open_lodems_sensor := "B18.4",
                top_sensor := "B18.0",
                mid_sensor := "S18.2",
                low_sensor := "DGI".GasketRampSqueeze_timer.Q,
                top_sensor_filter := "ALG".Auto_Sorting AND NOT "HS".Gasket_Ramp.Fault,
                QPLanksLayers := "DynamicLayer_CNTL_DB".ActualMaxHeight,
                CMD_On => "HS".Gasket_Ramp.setUp,
                CMD_Mid => "HS".Gasket_Ramp.setMid,
                CMD_Off => "HS".Gasket_Ramp.setDn,
                CMD_CloseLodems => "HS".Gasket_Lodems.OffCom,
                ENO => #_w2);
   #_s5time1 := S_ODT(T_NO := "Tag_95", S := #_w2 AND "FB_Ramp_DB".CMD_OpenLodems, TV := s5t#500ms, Q => #_w3);
   "HS".Gasket_Lodems.OnCom := #_w3;
END_REGION

REGION Network 66: Новый пакет
   RUNG wire#powerrail
      Contact( "DGI".btn_ResetUporLine.CMD_ON )
      S_SR(operand := #NewPacket, r1 := wire#w1)
   END_RUNG
   RUNG wire#powerrail
      Contact( #LiftDownTrig )
   END_RUNG wire#w1
   // the same network as SCL:
   IF "DGI".btn_ResetUporLine.CMD_ON THEN
       #NewPacket := TRUE;   // SR flip-flop
   END_IF;
   IF #LiftDownTrig THEN #NewPacket := FALSE; END_IF;
END_REGION

REGION Network 67: Синхронизация счетчиков с сервером
   RUNG wire#powerrail
      { S7_GenerateENO := "TRUE" } Move(in := #LayersCounter, out1 => "ServDB".NumLayerActual)
      { S7_GenerateENO := "TRUE" } Move(in := #BoardInLayerCounter, out1 => "ServDB".NumPlanksInLayerActual)
      { S7_GenerateENO := "TRUE" } Move(in := "ALG".LayerVolume, out1 => "ServDB".VLayerOk)
   END_RUNG
   // the same network as SCL:
   // ENO of a box is taken as its EN; it also drops when the box reports an error
   "ServDB".NumLayerActual := #LayersCounter;
   "ServDB".NumPlanksInLayerActual := #BoardInLayerCounter;
   "ServDB".VLayerOk := "ALG".LayerVolume;
END_REGION
END_FUNCTION_BLOCK

FUNCTION_BLOCK "Vibrator"
{ S7_Optimized_Access := 'FALSE' }
VERSION : 0.1
   VAR_INPUT 
      Signal : Bool;
   END_VAR

   VAR_OUTPUT 
      Out : Bool;
   END_VAR

   VAR 
      Signal_old : Bool;
   END_VAR


BEGIN
	IF (#Signal AND NOT #Signal_old) THEN
	    #Out := NOT #Out;
	END_IF;
	
	#Signal_old := #Signal;
END_FUNCTION_BLOCK

FUNCTION "WhatToDoWithNewSxema" : Void
{ S7_Optimized_Access := 'FALSE' }
VERSION : 0.1

BEGIN
	// зануляем счет на бобышках
	// 
	"UporPFM_DB".Counter := 0;
	
	// снимаем калибровку линейки
	// 
	"QueueController_DB".Calibrated := FALSE;
	
	// для режима из пакета  в пакет
	// 
	"DynamicLayer_CNTL_DB".notOk_Counter := 0;
END_FUNCTION

FUNCTION "GotNewLay" : Void
{ S7_Optimized_Access := 'FALSE' }
AUTHOR : Aspir
VERSION : 0.1
   VAR_INPUT 
      PlankL : Int;   // длина досок
      PlankW : Int;
      PlankT : Int;
   END_VAR

   VAR_IN_OUT 
      PlanksInLayer : Int;   // досок в текущем слое
      QPlanks_OK : Int;   // собрано досок в пакет
      Server_Volume : DInt;   // объем на серваке
      Layer_Volume : DInt;   // объем слоя
      Local_Volume : DInt;   // текущий насчитанный объем
   END_VAR


BEGIN
	// Добавляем слой к количеству хороших досок
	#QPlanks_OK := #QPlanks_OK + #PlanksInLayer;
	
	IF (#PlankL <> 0) THEN
	    #Layer_Volume := INT_TO_DINT(#PlanksInLayer) * INT_TO_DINT(#PlankL / 100) * INT_TO_DINT(#PlankW) * INT_TO_DINT(#PlankT);
	END_IF;
	
	
	// Добавляем значение объема слоя к текущему на ПЛК
	#Local_Volume := #Local_Volume + #Layer_Volume;
	
	// Обновляем показания на серваке
	// 
	#Server_Volume := #Local_Volume;
	
	#PlanksInLayer := 0;
	// Обнуляем счет объема слоя
	// 
	#Layer_Volume := 0;
END_FUNCTION

FUNCTION_BLOCK "KeyFazer_CNTL"
{ S7_Optimized_Access := 'FALSE' }
AUTHOR : Aspir
VERSION : 0.1
   VAR_INPUT 
      keyfazer_1 : Bool;   // сигнал кейфазера 1
      keyfazer_2 : Bool;   // сигнал кейфазера 2
      enableSensors : Bool;   // бит детектинга кейфазеров
   END_VAR

   VAR_OUTPUT 
      WheelChanged : Bool;   // колесо изменилось
      ActualWheelSig : Bool;   // сигнал с актуального колеса
      Chain : Bool;   // какой именно кейфазер сморим
      Window : Bool;   // окно между кейфазерами
      FaultKeyFazer : Bool;   // ошибка (померены две одинаковые цепи подряд)
   END_VAR

   VAR 
      active_wheel : Bool;   // текущее активное обмеряемое колесо
      validSig_old : Bool;
      changing_wheel : Bool;   // меняем показания реального колеса
      memento_act_wheel : Bool;   // запомненное колесо
      real_chain : Bool;   // реальная цепь
      AntiNoValidFront_timer {InstructionName := 'TON'; LibVersion := '1.0'; S7_SetPoint := 'False'} : TON;   // таймер защищающий от ложного фронта при включении двигателя
   END_VAR

   VAR_TEMP 
      stableRun : Bool;   // стабильный режим работы механизма
      faultSig : Bool;   // ошибочный сигнал с колес
      validSig : Bool;   // действительный сигнал с колеса
   END_VAR

   VAR CONSTANT 
      filterDelay : Time := T#200ms;   // через это время начнем видеть задние фронты колес
   END_VAR


BEGIN
	(*
	Кейфазеры работают по четверти периода оборота вала цепи с бобышками
	
	По их сигналу необходимо понимать когда должна обмерять линейка, проводить счет досок на слой ПФМ
	*)
	
	(* 
	//собираем все фронты сигналов и передние и задние
	//
	#p_front_1 := #keyfazer_1 AND NOT #keyfazer_1_old;
	#p_front_2 := #keyfazer_2 AND NOT #keyfazer_2_old;
	#n_front_1 := #keyfazer_1_old AND NOT #keyfazer_1;
	#n_front_2 := #keyfazer_2_old AND NOT #keyfazer_2;
	
	//сохраняем значения для ловли фронтов
	//
	#keyfazer_1_old := #keyfazer_1;
	#keyfazer_2_old:= #keyfazer_2; *)
	
	#AntiNoValidFront_timer(IN := #enableSensors,
	                        PT := #filterDelay);
	
	#stableRun := #AntiNoValidFront_timer.Q;
	
	#validSig := #active_wheel AND #keyfazer_1 OR NOT #active_wheel AND #keyfazer_2; // верный сигнал
	#faultSig := #active_wheel AND #keyfazer_2 OR NOT #active_wheel AND #keyfazer_1; //сигнал с ошибочным колесом
	
	// выходные сигналы
	// 
	#ActualWheelSig := #validSig;
	#Chain := #active_wheel;
	#Window := NOT (#keyfazer_1 OR #keyfazer_2);
	
	
	// для внутреннего контроля
	// 
	#real_chain := (#real_chain OR #keyfazer_1) AND NOT #keyfazer_2; // ВСЕГДА ПРЫГАЕТ МЕЖДУ ВЫСОКОЙ И НИЗКОЙ ЦЕПЬЮ
	
	//Если только поменял колесо и пошел сигнал ошибки значит чет не то и просто не будем менять еще раз колесо, это наверное дребезг
	//
	#changing_wheel := (#changing_wheel OR #WheelChanged) AND NOT (#validSig AND #stableRun);
	
	//крутим этот сигнал ровно один цикл
	#WheelChanged := FALSE;
	
	(*
	    Меняем колеcо по двум причинам:
	    1 - естественная:
	    транспортер едет и нужный сенсор дал задний фронт
	    2 - если вдруг по инерции проехали нужный нам задний фронт, то при включении двигателя проверим один раз ушли мы с датчика или нет
	*)
	
	IF (#stableRun AND ((NOT #validSig AND #validSig_old) OR (#faultSig AND NOT #changing_wheel))) THEN
	    #active_wheel := NOT #active_wheel;
	    #WheelChanged := TRUE;
	    #FaultKeyFazer := #real_chain <> #memento_act_wheel;
	    #memento_act_wheel := #real_chain;
	    
	    IF (#faultSig) THEN
	        #validSig := #active_wheel AND #keyfazer_1 OR NOT #active_wheel AND #keyfazer_2; // верный сигнал вычислим на всякий случай если сразу будет еще фронт (вряд ли нужно, такой большой инерции быть не может)
	    END_IF;
	END_IF;
	
	
	// для фронтов
	// 
	#validSig_old := #validSig;
END_FUNCTION_BLOCK

FUNCTION_BLOCK "KeyFazer_Counter"
{ S7_Optimized_Access := 'FALSE' }
AUTHOR : Aspir
VERSION : 0.1
   VAR_INPUT 
      NewWheel : Bool;   // сигнал о новом колесе
      RealChain : Bool;   // ныне проходящая цепь
      KeyFazerSignal : Bool;   // актуальный сигнал детекции
      PlankSensor : Bool;   // датчик-детектор доски на слой ПФМ
      AwaitedChain : Bool;   // ожидаемая цепь, на которой должны увидеть и посчитать доску
      Reset_count : Bool;   // сброс счета
      Reset_alarms : Bool;   // сброс ошибки
      PT : Int;   // пресет счета
   END_VAR

   VAR_OUTPUT 
      AlarmCount : Bool;   // ошибка счета
      Counted_one : Bool;   // доска была посчитана
   END_VAR

   VAR_IN_OUT 
      "Counter" : Int;   // счетчик
   END_VAR

   VAR 
      PlankCounted : Bool;   // доска посчитана на текущей цепи
      PlankSensor_old : Bool;
      PlankSensor_filter {InstructionName := 'TON'; LibVersion := '1.0'; S7_SetPoint := 'False'} : TON;
   END_VAR

   VAR_TEMP 
      Plank_front : Bool;
   END_VAR

   VAR CONSTANT 
      filterDelay : Time := T#100ms;
   END_VAR


BEGIN
	#Counted_one := FALSE;
	
	#PlankSensor_filter(IN:=#PlankSensor,
	                    PT:=#filterDelay);
	
	// Захватываем передний фронт доски каждый новый цикл на цепи по кейфазеру
	// 
	#Plank_front := #PlankSensor_filter.Q AND NOT #PlankSensor_old;
	
	// Ловим фронты
	#PlankSensor_old := #PlankSensor_filter.Q;
	
	//Если поймали фронт сигнала доски на данном периоде и на данном периоде она еще не была посчитана, значит все хорошо, увеличим счет
	IF (#Plank_front AND NOT #PlankCounted AND #Counter < #PT) THEN
	      #Counter := #Counter + 1;
	      #Counted_one := TRUE;
	END_IF;
	
	// Протестирую позже
	//#AlarmCount := (#AlarmCount OR (#PlankFront_catch_trig AND #RealChain <> #AwaitedChain));
	  
	#PlankCounted := (#PlankCounted OR #Plank_front) AND NOT #NewWheel;
	
	IF (#Reset_count) THEN
	    #Counter := 0;
	END_IF;
	
	
END_FUNCTION_BLOCK

FUNCTION_BLOCK "EvaluationZoneThrowOFF"
{ S7_Optimized_Access := 'FALSE' }
VERSION : 0.1
   VAR_INPUT 
      StartEvaluationArea : Bool;   // сигнал с датчика о наличии доски в начале зоны оценки
      EndEvaluationArea : Bool;   // сигнал с датчика конец зоны оценки
      DefectSignal : Bool;   // сигнал с кнопки брака
      MU_mode : Bool;   // местное управление сбросом в брак
      DropArea : Bool;   // сигнал с датчика перед сбросом
      Reset : Bool;   // сброс счетчиков
   END_VAR

   VAR_OUTPUT 
      DefectDrop_CMD_UP : Bool;   // команда на поднятие сбрасывателя
      DefectDrop_CMD_DOWN : Bool;   // команда на опускание сбрасывателя
      CommonAlarmEvaluationZone : Bool;   // авария на зоне оценки
      AlarmBoardNotExitFromZone : Bool;   // авария доска не покинула зону оценки
      FaultQueueOverflow : Bool;   // ошибка переполнения очереди
      FaultGhostBoard : Bool;   // ошибка "призрачная доска" (если почему-то указатель хвоста на нуле, при этом доска уехала с зоны оценки)
   END_VAR

   VAR 
      StartEvaluationArea_old : Bool;
      EndEvaluationArea_old : Bool;
      DropArea_old : Bool;
      CanEvaluate : Bool;   // доска почти наверное упала
      CMD_up_old : Bool;
      BoardIterator : Int;   // счетчик досок на зоне оценки (от первого датчика до сброса)
      SolutionQueue : Array[0..7] of Bool;   // очередь принятых решеий (брак - не брак)
      QueueCoded { ExternalAccessible := 'False'; ExternalVisible := 'False'; ExternalWritable := 'False'} AT SolutionQueue : Byte;
   END_VAR


BEGIN
	IF (#Reset AND (#CommonAlarmEvaluationZone)) THEN
	    IF (#FaultQueueOverflow OR #AlarmBoardNotExitFromZone) THEN
	        #BoardIterator := 0;
	        #FaultQueueOverflow := False;
	        #AlarmBoardNotExitFromZone := FALSE;
	        #CanEvaluate := FALSE;
	    END_IF;
	    #AlarmBoardNotExitFromZone := FALSE;
	
	    #FaultGhostBoard := FALSE;
	END_IF;
	
	#FaultQueueOverflow := #BoardIterator > 7;
	
	#CommonAlarmEvaluationZone := #AlarmBoardNotExitFromZone OR #FaultQueueOverflow OR #FaultGhostBoard;
	
	REGION Принятие решения на поштучке
	    
	    IF (#StartEvaluationArea AND NOT #StartEvaluationArea_old AND NOT #AlarmBoardNotExitFromZone) THEN
	        // передний фронт датчика начала зоны оценки 
	        #AlarmBoardNotExitFromZone := #CanEvaluate;
	        
	        #CanEvaluate := true;
	        
	        // пока запишем отрицательное решение оператора
	        // 
	        IF (NOT #FaultQueueOverflow) THEN
	            #SolutionQueue[#BoardIterator] := FALSE;
	        END_IF;
	    END_IF;
	    
	    IF (#DefectSignal AND #CanEvaluate AND NOT (#MU_mode OR #CommonAlarmEvaluationZone)) THEN
	        //Доска ушла с зоны оценки, можно фиксировать хвост (путем + 1) + снимаем флаг того, что доска оценивается
	        //
	        #SolutionQueue[#BoardIterator] := TRUE;
	    END_IF;
	    
	    IF ((NOT #EndEvaluationArea AND #EndEvaluationArea_old) AND #CanEvaluate AND NOT #AlarmBoardNotExitFromZone) THEN
	        // задний фронт конца зоны оценки либо нажата кнопка брак завершает задание для доски
	        // 
	        #BoardIterator := #BoardIterator + 1;
	        #CanEvaluate := FALSE;
	    END_IF;
	END_REGION
	
	REGION Движение сбрасывателя
	    
	    IF (#DropArea AND NOT #DropArea_old) THEN
	        // передний фронт датчика сброоса провоцирует pop первого элемента очереди
	        // 
	        #FaultGhostBoard := #BoardIterator = 0;
	        IF (NOT #FaultGhostBoard) THEN
	            
	            #DefectDrop_CMD_UP := #SolutionQueue[0];
	            #DefectDrop_CMD_DOWN := NOT #DefectDrop_CMD_UP;
	            
	            // двигаю очередь направо потому что биты перевернуты
	            #QueueCoded := SHR_BYTE(IN := #QueueCoded, N := 1); 
	            
	            //меняю указатель на хвост очереди
	            #BoardIterator := #BoardIterator - 1;
	        END_IF;
	        
	    END_IF;
	    
	END_REGION
	
	
	IF ((#CommonAlarmEvaluationZone OR #MU_mode) AND #DefectSignal) THEN
	    #DefectDrop_CMD_UP := NOT #DefectDrop_CMD_UP;
	    #DefectDrop_CMD_DOWN := NOT #DefectDrop_CMD_UP;
	END_IF;
	
	
	
	#CMD_up_old := #DefectDrop_CMD_UP;
	#StartEvaluationArea_old := #StartEvaluationArea;
	#EndEvaluationArea_old := #EndEvaluationArea;
	#DropArea_old := #DropArea;
END_FUNCTION_BLOCK

FUNCTION_BLOCK "SensorLine_Clogging"
{ S7_Optimized_Access := 'FALSE' }
VERSION : 0.1
   VAR_INPUT 
      KeyFazer : Bool;
      Reset : Bool;
      SensLine_sig : Word;
   END_VAR

   VAR_OUTPUT 
      AlarmSensor_dirty : Array[0..15] of Bool;
      AlarmArray { ExternalAccessible := 'False'; ExternalVisible := 'False'; ExternalWritable := 'False'} AT AlarmSensor_dirty : Word;
      AlarmSensorLine : Bool;
   END_VAR

   VAR 
      KeyFazer_old : Bool;
      LowDetected : Word;
      Ala : Word;
   END_VAR

   VAR_TEMP 
      front : Bool;
   END_VAR

   VAR CONSTANT 
      SensorQuantity : Int := 15;
   END_VAR


BEGIN
	#front := (#KeyFazer AND NOT #KeyFazer_old)(* OR (NOT #KeyFazer AND #KeyFazer_old) *);
	
	IF (#front) THEN
	    // проверяем, были ли все сигналы хоть раз False
	  
	    #AlarmArray := #AlarmArray OR NOT #LowDetected;
	    
	    #AlarmSensorLine := #AlarmSensorLine OR (#AlarmArray AND 2#1111_1111_0111_1111) <> 16#0;
	    //обнуляем триггеры, начинаем новый цикл
	    #LowDetected := 16#0;
	    
	ELSE
	    // в противном случае смотри за тем чтобы хоть раз были в нуле сенсоры
	    //
	    #LowDetected := #LowDetected OR NOT #SensLine_sig;
	END_IF;
	
	IF (#Reset AND #AlarmSensorLine) THEN
	    #AlarmArray := 2#0000_0000_0000_0000;
	    #AlarmSensorLine := FALSE;
	END_IF;
	
	#Ala := #AlarmArray;
	
	
	// ловим фронты
	//
	#KeyFazer_old := #KeyFazer;
END_FUNCTION_BLOCK

FUNCTION_BLOCK "SensLine_SigAdapter"
{ S7_Optimized_Access := 'FALSE' }
VERSION : 0.1
   VAR_INPUT 
      InputSig : Word;
      InputArr { ExternalAccessible := 'False'; ExternalVisible := 'False'; ExternalWritable := 'False'} AT InputSig : Array[0..15] of Bool;
   END_VAR

   VAR_OUTPUT 
      OutputSig : Word;
      OutputArr { ExternalAccessible := 'False'; ExternalVisible := 'False'; ExternalWritable := 'False'} AT OutputSig : Array[0..15] of Bool;
   END_VAR

   VAR 
      timer_18 {InstructionName := 'TON'; LibVersion := '1.0'; S7_SetPoint := 'False'} : TON;
      timer_42 {InstructionName := 'TON'; LibVersion := '1.0'; S7_SetPoint := 'False'} : TON;
      timer_48 {InstructionName := 'TON'; LibVersion := '1.0'; S7_SetPoint := 'False'} : TON;
      timer_51 {InstructionName := 'TON'; LibVersion := '1.0'; S7_SetPoint := 'False'} : TON;
      timer_57 {InstructionName := 'TON'; LibVersion := '1.0'} : TON;
   END_VAR

   VAR CONSTANT 
      delayFilter : Time := T#100ms;
   END_VAR


BEGIN
	//просто копирование до фильтрации отдельных битов
	//
	#OutputSig := #InputSig;
	
	//Блок фильтрации
	// 1.8 m
	#timer_18(IN:=#InputArr[0],
	          PT:=#delayFilter);
	
	#OutputArr[0] := #timer_18.Q;
	
	// 4.2 m
	#timer_42(IN := #InputArr[8],
	          PT := #delayFilter);
	
	#OutputArr[8] := #timer_42.Q;
	
	// 4.8 m
	#timer_48(IN := #InputArr[10],
	          PT := #delayFilter);
	
	#OutputArr[10] := #timer_48.Q;
	
	// 5.1 m
	#timer_51(IN := #InputArr[11],
	          PT := #delayFilter);
	
	#OutputArr[11] := #timer_51.Q;
	
	// 5.7 m
	#timer_57(IN := #InputArr[13],
	          PT := T#150ms);
	
	#OutputArr[13] := #timer_57.Q;
	
END_FUNCTION_BLOCK

FUNCTION_BLOCK "FB_SensLine"
{ S7_Optimized_Access := 'FALSE' }
AUTHOR : Aspir
VERSION : 0.1
   VAR_INPUT 
      CutPlankData : Bool;   // сигнал на анализ данныз и выдаче результатов
      CollectData : Bool;   // собирать данные под линейкой
      ActualChain : Bool;   // текущая цепь для измерений
      EnableSensors : Bool;   // включить датчики на измерение
      SensData : Word;   // данные с датчиков в формате Word (по порядку)
      SensDataArray { ExternalAccessible := 'False'; ExternalVisible := 'False'; ExternalWritable := 'False'} AT SensData : Array[0..15] of Bool;   // в виде массива булов
      SensDataByte { ExternalAccessible := 'False'; ExternalVisible := 'False'; ExternalWritable := 'False'} AT SensData : Array[0..1] of Byte;   // массив байтов
      SensQuantity : Int;   // Количество датчиков
      MinLength : Int;   // минимальная длина, мм
      SensOffset : Int;   // расстояние между датчиками, мм
   END_VAR

   VAR_OUTPUT 
      Done : Bool;   // сделал измерение
      Hole : Bool;   // ничего нет, имеем дырку
      Chain : Bool;   // на какой цепи измерил (0 - на низкой, 1 - на высокой)
      Length : Int;   // измеренная длина
   END_VAR

   VAR 
      memento_chain : Bool;
      sensor_triggers : Array[0..15] of Bool;
      sensor_triggers_WORD { ExternalAccessible := 'False'; ExternalVisible := 'False'; ExternalWritable := 'False'} AT sensor_triggers : Word;
      sensor_triggers_INT { ExternalAccessible := 'False'; ExternalVisible := 'False'; ExternalWritable := 'False'} AT sensor_triggers : Int;
   END_VAR

   VAR_TEMP 
      real_index : Int;   // реальный индекс с учетом обратного порядка байтов
      index : Int;
      tmp_restruct : Word;   // слово для реструктуризации
   END_VAR


BEGIN
	// СБрасываем флаг Done чтобы он висел всего одлин цикл после измерения
	// 
	#Done := FALSE;
	#Hole := FALSE;
	
	// Получили разрешение на триггер сигналов - за работу
	// В цикле проверяем каждый датчик
	// 
	IF (#CollectData AND #EnableSensors) THEN
	    // TESTED!!
	    // реструктурируем данные для удобного расчета
	    // Байты в слове переставляются наоборот
	    // 1111000_00001111 -> 00001111_1111000
	    #tmp_restruct := SHL_WORD(IN:= BYTE_TO_WORD(#SensDataByte[1]), N := 8) OR BYTE_TO_WORD(#SensDataByte[0]);
	    #tmp_restruct := #tmp_restruct AND INT_TO_WORD(WORD_TO_INT(SHL_WORD(IN := DINT_TO_WORD(16#1), N := #SensQuantity)) - 1);
	    #sensor_triggers_WORD := #sensor_triggers_WORD OR #tmp_restruct;
	    
	    
	    // Not optimized
	    (* FOR #index := 0 TO #SensQuantity - 1 DO
	        // вычислим реальный индекс в массиве
	        // Аналогично в блоке FB_SetGaskets
	        #real_index := #index + 7 - 2 * (#index MOD 8);
	        // триггерим показания
	        #sensor_triggers[#index] := #sensor_triggers[#index] OR #SensDataArray[#real_index]; 
	    END_FOR; *)
	    
	END_IF;
	
	// снимаем сливки (длину) по заднему фронту хоть одного из колес
	// 
	IF (#CutPlankData) THEN
	    // указываю, на какой цепи померил
	    // 
	    #memento_chain := #Chain;
	    #Chain := #ActualChain;
	    // если цепь та же самая явно что-то не то, выходим
	    IF (#Chain = #memento_chain) THEN
	        "ALG".TestCounter2 := "ALG".TestCounter2 + 1;
	        RETURN;
	    END_IF;
	    
	     // Вычисляем длину
	    // 
	    IF (#sensor_triggers[8]) THEN
	        // TESTED!!
	        // Вычисление длины
	        #Length := #MinLength + #SensOffset * TRUNC_INT(LN(INT_TO_REAL(#sensor_triggers_INT)) / LN(2.0));
	        
	        (* // Not optimized
	        // Далее проходим по массиву, накапливая длину по offset
	        #Length := #MinLength;
	        #index := 14;
	        
	        WHILE (#sensor_triggers[#index] AND (#index >= 16 - #SensQuantity))DO
	            #Length := #Length + #SensOffset;
	            #index := #index - 1;
	        END_WHILE; *)
	        
	        #Done := TRUE;
	    ELSE
	        #Length := 0;
	        #Done := FALSE;
	        
	        #Hole := TRUE;
	    END_IF;
	    
	    // сбрасываю триггеры всех датчиков
	    #sensor_triggers_WORD := 16#0;
	    
	END_IF;
END_FUNCTION_BLOCK

FUNCTION_BLOCK "QueueController"
{ S7_Optimized_Access := 'FALSE' }
AUTHOR : Aspir
VERSION : 0.1
   VAR_INPUT 
      Reset : Bool;   // сброс ошибки
      ResetSxema : Bool;   // сброс калибровки
      NoChessLayout : Bool;   // не нужна ли шахматка при укладке
      CheckPlankL : Bool;   // нужна ли проверка длины доски
      ChainInd : Bool;   // цепь на которой было измерение
      Hole : Bool;   // Дырка под линейкой
      Done : Bool;   // Линейка сделала измерение длины
      Length : Int;   // Измеренная длина
      CheckL : Int;   // Проверяемая длина
      PT : Int;   // досок на слой
      plankW : Int;   // ширина доски
      plankT : Int;   // толщина доски
      OffsetBB : Int;   // сдвиг между попом и пушем
   END_VAR

   VAR_OUTPUT 
      CommonSxemaAlarm : Bool;   // общая авария схемы
      AlarmNotAwaitableBoard : Bool;   // авария лишняя доска в схеме
      AlarmNotValidHole : Bool;   // авария нет дырки между схемами
      AlarmCount : Bool;   // ошибка счета на слой
      AlarmWrongLength : Bool;   // ошибка неверная длина
      Hint_1 : Bool;   // уточнение к аварии 1 (после следующей доски должна быть дырка)
      Hint_2 : Bool;   // уточненная авария 2 (выкидываем доску)
      Hint_3 : Bool;   // уточнение по ожидаемой цепи
      CorrectingCounters : Bool;   // Состояние корректировки счетчиков упоров
      CorrectCounters : Bool;   // корректировка счета
      CorrectWheel : Bool;   // корректировка колеса (высокое или низкое)
      GettingLastLay : Bool;   // Сейчас собираю последний слой на пакет
      CurrentLayCounter : Int;   // текущий счетчик для проверки схемы слоя
   END_VAR

   VAR_IN_OUT 
      BoardsInLay_counter : Int;   // счетчик досок на слой
      Layer_Volume { ExternalAccessible := 'False'; ExternalVisible := 'False'; ExternalWritable := 'False'} : DInt;   // объем  текущего слоя, м3
   END_VAR

   VAR 
      Calibrated : Bool;   // калибровка решателя
      AwaitedChain : Bool;   // Ожидаемая по высоте цепь
      AwaitEmptySpace : Bool;   // Ожидание пустого места
      ProcessedError : Bool;   // ошибка обработана
      CanPutBoardHoleBefore : Bool;   // можно пололжить доску в пустоту вперед
      LugCounter : Int;
      Data { S7_SetPoint := 'False'} : Array[0..#QueueSize] of "PlankOnChain";   // основные данные о досках
   END_VAR

   VAR_TEMP 
      ValidSpace : Bool;   // валидное поле для потенциальной доски
      WrongLength : Bool;   // ошибка некорректная длина доски
      Pop_Push : Bool;   // заполнить/вытащить
      index : Int;   // индекс для копирования
      PlankVolume : DInt;   // объем досточки
   END_VAR

   VAR CONSTANT 
      QueueSize : Int := 15;   // размер очереди
      CorrectingOffset : Int := 7;   // количество бобышек, которое проходит транспортер для корректировки
   END_VAR


BEGIN
	#CorrectCounters := FALSE;
	    
	REGION Проверка длины 
	    // Проверка длины
	    // 
	    #WrongLength := #CheckPlankL AND #Done AND #Length <> #CheckL;
	        
	    #AlarmWrongLength := (#AlarmWrongLength OR #WrongLength);
	END_REGION
	    
	    
	REGION Логика проверки схемы укладки досок
	    #Pop_Push := #Done OR #Hole;
	        
	    IF (#Calibrated) THEN
	        IF (NOT #AwaitEmptySpace) THEN
	                        
	                    #ValidSpace := #AwaitedChain = #ChainInd;
	                        
	                    IF (#Hole OR #AlarmWrongLength) THEN
	                        // Если пришла дырка считаем запас
	                        // будет нужно для выкидывания хинта операторам
	                        // Если доска некорректной длины не будем считать это за дырку
	                        // запустим восстановление счета упоров
	                        // 
	                        #CanPutBoardHoleBefore := #ValidSpace AND NOT #AlarmWrongLength;
	                            
	                    ELSIF (#Done) THEN
	                        // Если пришла нормальная по длине доска и не дырка
	                        // 
	                        IF (#ValidSpace OR #NoChessLayout) THEN
	                                // сбрасываем флаг валидности цепи для укладки потенциально неправильной доски
	                                // 
	                                #CanPutBoardHoleBefore := FALSE;
	                               
	                                 // меняем ожидаемую цепь
	                                 #AwaitedChain := NOT #AwaitedChain;
	                                    
	                                 // увеличиваем счет
	                                 // И проверяем, надо ли дальше ждать пустое место
	                                 #CurrentLayCounter := #CurrentLayCounter + 1;
	                                    
	                                 // Проверяем, набрали ли на слой доски
	                                 // Если набрали просто выставляем ожидание на дырку
	                                 #AwaitEmptySpace := #CurrentLayCounter = #PT;
	                                   
	                        ELSE
	                            // Если случилось что-то не то
	                            //  выкидываем ошибку о том что пришла доска но не на той цепи
	                            #AlarmNotAwaitableBoard := NOT #ValidSpace;
	                                    
	                        END_IF;
	                        
	                    END_IF;
	                           
	        ELSE
	        // Ожидаем пустое место
	                    IF (#Pop_Push) THEN
	                         //НО пришла доска, выкинем ошибку
	                         #AlarmNotValidHole := #Done;
	                         // Была ожидаемая дырка все гуд, можно сбросить все необходимое
	                         
	                         //Если ожидали дырку и получили ее, просто меняем ожидаемую доску на обратную от предыдущего слоя
	                         IF (#PT MOD 2 = 0) THEN
	                              #AwaitedChain := NOT #AwaitedChain;
	                         END_IF;
	                                
	                         #CurrentLayCounter := 0;
	                         //Говорим, что данная образование не может служить для доски, нельзя положить на данную пустую цепь
	                         #CanPutBoardHoleBefore := FALSE;
	                            
	                         // Выходим отсюда
	                         #AwaitEmptySpace := FALSE;
	                                
	                    END_IF;
	                       
	        END_IF;
	    END_IF;
	END_REGION
	        
	    REGION Обработка ошибок и выкидывание хинтов
	        
	        IF (#AlarmNotAwaitableBoard AND NOT #ProcessedError) THEN
	            //ошибка ДОСКА ПРИШЛА НЕ НА ТОЙ ЦЕПИ
	            //Эта ошибка выползает только в режиме раскатки
	            //При этой ошибке доска считается линейкой и записывается в очередь, поэтому ее важно просто положить на нужную цепь соответсвенно низкую или высокую после линейки
	            // 
	            // 1 вариант решения проблемы
	            // Если у нас есть лишная пустота выкидываем сообщение о том чтобы перекинули доску на соседнюю высокую или низкую цепь, из системы доску НЕ удаляем
	            // 2 вариант 
	            // Если нет лишних пустот удаляем доску из системы и говорим убрать ее нафиг с линии
	            // 
	            #ProcessedError := TRUE;
	            // выдаем хинт
	            // 
	            #Hint_1 := #CurrentLayCounter = #PT - 1; // последняя доска в слое
	            //#Hint_2 := true;
	            
	            #Hint_2 := NOT #CanPutBoardHoleBefore; // если можем подложить доску вперед, просто даем системе ее учесть
	            
	             IF (#CanPutBoardHoleBefore) THEN
	                // Если возможен вариант с перекидыванием доски вперед на бобышку, используем его, учтем доску в системе
	                // сбрасываем флаг валидности цепи для укладки потенциально неправильной доски
	                // 
	                #CanPutBoardHoleBefore := FALSE;
	                
	                
	                // увеличиваем счет
	                // И проверяем, надо ли дальше ждать пустое место
	                // так как дырка образуется сама собой проверяем, не можем ли просто начать счет заново
	                // 
	                IF (#Hint_1) THEN
	                    // это будет последняя доска на слой плюс получили дырку
	                    // ПОКА ЧТО ЭТО ДУБЛИРОВАНИЕ КОДА, НЕТ ВРЕМЕНИ ПЕРЕДЕЛАТЬ!
	                    
	                    //Если ожидали дырку и получили ее, просто меняем ожидаемую доску на обратную от предыдущего слоя
	                    IF (#PT MOD 2 <> 0) THEN
	                        #AwaitedChain := NOT #AwaitedChain;
	                    END_IF;
	                    
	                    #CurrentLayCounter := 0;
	                    
	                ELSE
	                    // если доска не последняя в слой
	                    // 
	                    // меняем ожидаемую цепь
	                    #AwaitedChain := NOT #AwaitedChain; 
	                    
	                    // увеличиваем счет
	                    // И проверяем, надо ли дальше ждать пустое место
	                    #CurrentLayCounter := #CurrentLayCounter + 1;
	                    
	                END_IF;
	     
	            END_IF; 
	            
	            #Hint_3 := #AwaitedChain; // хинт на ожидаемую цепь
	            
	        ELSIF (#AlarmNotValidHole AND NOT #ProcessedError) THEN
	            //ошибка ОЖИДАЛАСЬ ДЫРКА А ПРИШЛА ДОСКА НА ЦЕПИ
	            //Эту доску по-любому будем выкидывать, поэтому вопрос решается легко
	            #ProcessedError := TRUE;
	            #Hint_2 := TRUE;
	            // Дополнительно скажем заранее, какая цепь должна быть следующей
	            #Hint_3 := #AwaitedChain;
	        END_IF;
	        
	    END_REGION
	    
	    
	    REGION Корректировка счетчиков упоров
	        // Statement section REGION
	        // Ждем прохождения бобышек между плавниками и линейкой, корректируем счет на упорах перед бобышками
	        // 
	        IF (#CorrectingCounters AND (#Done OR #Hole)) THEN
	                #LugCounter := #LugCounter + 1;
	                
	                #CorrectWheel := #AwaitedChain;
	                
	                #CorrectCounters := #LugCounter = #CorrectingOffset;
	                
	                #CorrectingCounters := NOT #CorrectCounters;
	        END_IF;
	        
	    END_REGION
	    
	    REGION Калибруем решатель
	        // Если супер-проверщик по линейке не откалиброван, не знает, какая первая доска должна прийти, обязательно его калибруем по первой пришедшей "живой" доске
	        // Занимаемся проверкой шахматки в соответствующем режиме
	        IF (#Done AND NOT #Calibrated AND NOT #AlarmWrongLength) THEN
	            #Calibrated := TRUE;
	            // Поняли, какую цепь ожидаем следующей
	            #AwaitedChain := NOT #ChainInd;
	            // НЕ ожидаем пустое место, вряд ли у них пакет из одной доски собирается
	            #AwaitEmptySpace := FALSE;
	            // Добавили доску к счету
	            // 
	            #CurrentLayCounter := 1;
	            // Счет слоев обнуляем
	            // 
	            #GettingLastLay := FALSE;
	            
	            //После сброса запускаем задание на коррекцию счета упоров
	            #CorrectingCounters := TRUE;
	            #LugCounter := 0;
	        END_IF;
	        
	    END_REGION
	    
	    REGION Сброс калибровки
	        // Statement section REGION
	        
	        IF (#ResetSxema) THEN
	            #Calibrated := FALSE;
	        END_IF;
	    END_REGION
	    
	    // Здесь логика заполнения и опустошения очереди
	    // 
	    REGION Push and Pop
	        
	        IF (#Pop_Push) THEN
	            // Если чет было добавим это к объему и количеству досок на слой
	            // 
	            #AlarmCount := (#AlarmCount OR (#Data[0].NoEmpty AND #BoardsInLay_counter >= #PT));
	            
	            IF (#Data[0].NoEmpty AND #BoardsInLay_counter < #PT) THEN
	                // Считаем объем слоя! на вилах
	                #PlankVolume := INT_TO_DINT(#plankT) * INT_TO_DINT(#plankW) * INT_TO_DINT(#Data[0].Length) / 100;
	                #Layer_Volume := #Layer_Volume + #PlankVolume;
	                #BoardsInLay_counter := #BoardsInLay_counter + 1;
	                
	            END_IF;
	            
	            
	            // сдвиг всех значений на единицу
	            FOR #index := 0 TO #OffsetBB - 1 DO
	                // с первого до длины - 1
	                // 
	                #Data[#index] := #Data[#index + 1];
	            END_FOR;
	            
	            IF (#AlarmNotAwaitableBoard AND NOT #Hint_2) THEN
	                // Если была авария переложить доску на соседнюю бобышку, заполним предыдущее значение
	                // 
	                #Data[#OffsetBB - 1] := "PlankChain"(Chain := NOT #ChainInd, Empty := FALSE, Length := #Length);
	            END_IF;
	            // Заполнение очереди померенной доской
	            #Data[#OffsetBB] := "PlankChain"(Chain := #ChainInd, Empty:= #Hole OR #AlarmNotAwaitableBoard OR #AlarmNotValidHole OR #AlarmWrongLength, Length := #Length);
	
	        END_IF;
	    END_REGION
	    
	    REGION Сброс ошибок
	        // Statement section REGION
	        IF (#Reset AND (#AlarmNotAwaitableBoard OR #AlarmNotValidHole OR #AlarmWrongLength OR #AlarmCount)) THEN
	            //После сброса запускаем задание на коррекцию счета упоров
	            #CorrectingCounters := #AlarmNotAwaitableBoard OR #AlarmNotValidHole OR #AlarmWrongLength;
	            #LugCounter := 0;
	            
	            #AlarmNotAwaitableBoard := False;
	            #AlarmNotValidHole := FALSE;
	            #AlarmWrongLength := FALSE;
	            #AlarmCount := FALSE;
	            
	            #CommonSxemaAlarm := FALSE;
	            #Hint_3 := FALSE;
	            #Hint_2 := FALSE;
	            #Hint_1 := FALSE;
	            
	            #ProcessedError := FALSE;
	            
	            
	        END_IF;
	        
	        #CommonSxemaAlarm := #CommonSxemaAlarm OR (#AlarmNotAwaitableBoard OR #AlarmNotValidHole OR #AlarmCount OR #AlarmWrongLength);
	    END_REGION
	
	
END_FUNCTION_BLOCK

FUNCTION "PlankChain" : "PlankOnChain"
{ S7_Optimized_Access := 'FALSE' }
VERSION : 0.1
   VAR_INPUT 
      Chain : Bool;
      Empty : Bool;
      Length : Int;
   END_VAR


BEGIN
	#PlankChain.Chain := #Chain;
	#PlankChain.NoEmpty := NOT #Empty;
	#PlankChain.Length := #Length;
END_FUNCTION

FUNCTION_BLOCK "UporPFM"
{ S7_Optimized_Access := 'FALSE' }
VERSION : 0.1
   VAR_INPUT 
      firstWheel : Bool;
      secondWheel : Bool;
      boardSensorClose : Bool;   // сигнал о наличии доски под забором
      boardSensorFar : Bool;
      readyStartPacket : Bool;   // сигнал начала задания
      stopTask : Bool;   // бит на окончание задания (дособрать последний слой)
      NoChessLayout : Bool;   // не нужна раскатка
      MuchBoards : Bool;   // кнопка набора ковра
      ResetFaults : Bool;   // сброс ошибок
      Correcting : Bool;
      CorrectCounters : Bool;   // сброс счета
      CorrectedWheel : Bool;
      BoardsInLay : Int;   // досок в слое
      Length : Int;   // длина доски
      CorrectedCounter : Int;
   END_VAR

   VAR_OUTPUT 
      CMD_Up : Bool;
      CMD_Down : Bool;
      CommonAlarm : Bool;   // общая ошибка на упорах
      AlarmGidra : Bool;   // Ошибка сработки упоров
      AlarmWarpingBoard : Bool;   // Ошибка перекоса доски
   END_VAR

   VAR 
      firstWheel_old : Bool;
      secondWheel_old : Bool;
      muchBoards_old : Bool;
      boardSensor_old : Bool;
      currentSelectedWheel : Bool;
      needWork : Bool;
      haveTask : Bool;
      Skip : Bool;
      DenyAlarm : Bool;
      helper : Bool;
      "Counter" : Int;
      notAwaitableBoard_timer {InstructionName := 'TON'; LibVersion := '1.0'; S7_SetPoint := 'False'} : TON;
      notStableLayer_timer {InstructionName := 'TOF'; LibVersion := '1.0'} : TOF;
      StableLayer_timer {InstructionName := 'TON'; LibVersion := '1.0'} : TON;
   END_VAR

   VAR_TEMP 
      currentWheel_sig : Bool;
      currentWheel_sig_old : Bool;
      NoNeedSkip : Bool;
      boardSignal : Bool;   // обобщенный сигнал с датчиков доски
   END_VAR


BEGIN
	//корректировка счета и колеса
	//
	IF (#CorrectCounters) THEN
	    IF (#CorrectedCounter = #BoardsInLay) THEN
	        #Counter := 0;
	    ELSE
	        #Counter := #CorrectedCounter;
	    END_IF;
	    #currentSelectedWheel := #CorrectedWheel;
	END_IF;
	
	//выбор сигнала по колесу
	IF (#currentSelectedWheel) THEN
	    #currentWheel_sig := #firstWheel;
	    #currentWheel_sig_old := #firstWheel_old;
	ELSE
	    #currentWheel_sig := #secondWheel;
	    #currentWheel_sig_old := #secondWheel_old;
	END_IF;
	
	// новое задание (новый пакет)
	IF (NOT #haveTask AND #readyStartPacket) THEN
	    #haveTask := true;
	    #Skip := FALSE;
	END_IF;
	
	// пока так, позже добавлю логику и фильтры
	// Сигнал наличия доски
	#boardSignal := #boardSensorClose AND (#boardSensorFar OR #Length < 3000);
	
	
	// начинаем работу упоров либо если опер нажал кнопочку, либо если работаем без раскатки, там пофиг
	#needWork := (#needWork OR (#MuchBoards AND NOT #muchBoards_old)) AND NOT #Correcting;
	
	//Надо делать двойную дырку
	//
	#NoNeedSkip := NOT #Skip OR #NoChessLayout;
	
	#notStableLayer_timer(IN := #boardSignal,
	                      PT := T#400ms);
	
	#StableLayer_timer(IN:=#boardSignal,
	                   PT:=T#150ms);
	
	#notAwaitableBoard_timer(IN := #boardSensorClose OR #boardSensorClose,
	                         PT := T#150ms);
	
	IF (#ResetFaults) THEN
	    #AlarmGidra := FALSE;
	    #AlarmWarpingBoard := FALSE;
	
	END_IF;
	
	
	IF (#needWork AND #haveTask) THEN
	    // всегда смотрим за стабильностью сигнала с датчиков досок, он должен быть постоянным
	    //
	    IF (#DenyAlarm) THEN
	        IF (#boardSignal) THEN
	            #DenyAlarm := FALSE;
	        END_IF;
	    ELSIF (NOT #notStableLayer_timer.Q AND #CMD_Down) THEN
	        // поднимаем упоры и кричим о том что что-то не так
	        // 
	        #CMD_Up := True;
	        #CMD_Down := FALSE;
	        
	        #needWork := FALSE;
	        
	        #AlarmWarpingBoard := #boardSensorClose OR #boardSensorFar;
	        
	    END_IF;
	    
	    // По переднему фронту текущего сигнала опускаем упоры, даем шанс доске упасть в нужное место
	    IF (#currentWheel_sig AND NOT #currentWheel_sig_old AND #NoNeedSkip) THEN
	        // Запрещаю выброс аварии если до этого были вверху
	        // 
	        #DenyAlarm := #CMD_Up;
	        
	        #CMD_Down := TRUE;
	        #CMD_Up := FALSE;
	            
	            
	    END_IF;
	    
	    // По заднему фронту 
	    IF (NOT #currentWheel_sig AND #currentWheel_sig_old) THEN
	        IF (#NoNeedSkip) THEN
	            IF (#StableLayer_timer.Q) THEN
	                // Если сигнал с датчика доски есть, считаем, что заберем с текущего колеса доску и можно укладывать на следующую
	                // Соответсвенно ничего не делаем с упорами, все гуд
	                #currentSelectedWheel := NOT #currentSelectedWheel;
	                
	                #Counter := #Counter + 1;
	                
	                IF (#Counter = #BoardsInLay) THEN
	                    // Если досчитали доски до нужного числа и нужен пробел, надо еще раз поменять колесо и поднять таки упоры
	                    // 
	                    #Skip := #BoardsInLay MOD 2 <> 0;
	                    
	                    IF (NOT #Skip OR #NoChessLayout) THEN
	                        
	                        #currentSelectedWheel := NOT #currentSelectedWheel;
	                    END_IF;
	                    
	                    #CMD_Up := True;
	                    #CMD_Down := FALSE;
	                    
	                    #Counter := 0;
	                    
	                    // Если приказали дособирать этот слой и встать, так и делаем
	                    // 
	                    #haveTask := NOT #stopTask;
	                END_IF;
	                
	            ELSE
	                // Доски не было, поднимаем упоры, должны уложить на наше колесо
	                #CMD_Up := True;
	                #CMD_Down := FALSE;
	                
	                // снова ждем хорошего ковра перед упорами
	                #needWork := FALSE;
	            END_IF;
	        ELSE
	            #Skip := FALSE;
	        END_IF;
	    END_IF;
	ELSE
	    // если не работаем, поднимаем упоры и ждем!
	    // 
	    
	    IF (#notAwaitableBoard_timer.Q AND NOT #boardSensor_old) THEN
	        #AlarmGidra := TRUE;
	    END_IF;
	    
	    #CMD_Up := True;
	    #CMD_Down := FALSE;
	END_IF;
	
	
	#CommonAlarm := #AlarmGidra OR #AlarmWarpingBoard;
	    
	#firstWheel_old := #firstWheel;
	#secondWheel_old := #secondWheel;
	#muchBoards_old := #MuchBoards;
	#boardSensor_old := #notAwaitableBoard_timer.Q;
END_FUNCTION_BLOCK

FUNCTION_BLOCK "DynamicLayer_CNTL"
{ S7_Optimized_Access := 'FALSE' }
AUTHOR : Aspir
VERSION : 0.1
   VAR_INPUT 
      NewPack : Bool;   // начало нового пакета
      EnableDynamicLayer : Bool;   // включение функции динамических слоев
      NotOkSensor : Bool;   // счетчик плохих досок
      PackMaxHeight : Int;   // максимальная высота пакета
      BoardsInLay : Int;   // досок на слой
      BoardsInCurrentPack : Int;   // Всего досок в пакете
   END_VAR

   VAR_OUTPUT 
      ActualMaxHeight : Int;   // текущее скорректированное число слоев
   END_VAR

   VAR 
      NotOkSensor_old : Bool;
      notOk_Counter : Int;   // счетчик плохих досок
   END_VAR


BEGIN
	
	IF NOT #EnableDynamicLayer THEN
	    // Если не нужна данная функция и работаем на потоке, не будем ничего считать и просто отошлем параметр пакета
	    // 
	    #notOk_Counter := 0;
	    #ActualMaxHeight := #PackMaxHeight;
	ELSE
	    IF (#NotOkSensor AND NOT #NotOkSensor_old) THEN
	        #notOk_Counter := #notOk_Counter + 1;
	    END_IF;
	    
	    #ActualMaxHeight := DINT_TO_INT(CEIL(INT_TO_REAL(#BoardsInCurrentPack - #notOk_Counter) / #BoardsInLay));
	    
	    IF (#ActualMaxHeight > #PackMaxHeight) THEN
	        #ActualMaxHeight := #PackMaxHeight;
	    END_IF;
	END_IF;
	
	
	(* // Кнопка новый пакет
	IF (#NewPack) THEN
	    #notOk_Counter := 0;
	END_IF; *)
	
	// Ловим фронты
	#NotOkSensor_old := #NotOkSensor;
	
	
	
END_FUNCTION_BLOCK

FUNCTION_BLOCK "FB_Ramp"
{ S7_Optimized_Access := 'FALSE' }
VERSION : 0.1
   VAR_INPUT 
      add_lay : Bool;   // еще слой
      to_empty : Bool;   // ложементы очищены
      new_packet : Bool;   // новый пакет
      push_packet : Bool;   // форсим пакет
      pick_gaskets : Bool;   // нужен слой прокладок
      gaskets_acquire : Bool;   // можно забирать с крюков
      gaskets_released : Bool;   // можно опускать
      gaskets_busy : Bool;
      mode_no_gasket : Bool;   // режим без прокладок
      forks_start_sensor : Bool;
      open_lodems_sensor : Bool;
      top_sensor : Bool;
      mid_sensor : Bool;
      low_sensor : Bool;
      top_sensor_filter : Bool;
      QPLanksLayers : Int;
   END_VAR

   VAR_OUTPUT 
      carousel_full_reset : Bool;
      sig_carousel_release_gaskets : Bool;
      make_gasket_layer : Bool;
      lock_forks : Bool;
      lock_carousel : Bool;
      last_lay : Bool;
      down_working : Bool;
      ramp_not_up : Bool;
      ramp_not_down : Bool;
      CMD_On : Bool;
      CMD_Mid : Bool;
      CMD_Off : Bool;
      CMD_OpenLodems : Bool;
      CMD_CloseLodems : Bool;
      layer_holded : Int;
   END_VAR

   VAR 
      s_busy : Bool;
      s_lay_cmd_permission : Bool;
      _State : Int;
   END_VAR

   VAR CONSTANT 
      STATE_INIT : Int := 0;
      STATE_AWAIT : Int := 3;
      STATE_RELEASE_GASKETS : Int := 5;
      STATE_OPENING_LODEMS : Int := 6;
      STATE_ACQUIRE_GASKETS : Int := 7;
      STATE_WAIT_RELEASE : Int := 8;
      STATE_PUSHING_PACKET : Int := 9;
   END_VAR


BEGIN
	
	#ramp_not_up := (#ramp_not_up OR (#mid_sensor OR #low_sensor)) AND NOT #top_sensor;
	#ramp_not_down := (#ramp_not_down OR (#mid_sensor OR #top_sensor)) AND NOT #low_sensor;
	
	#carousel_full_reset := FALSE;
	
	IF (#to_empty) THEN
	    #s_busy := FALSE;
	END_IF;
	
	IF (#add_lay) THEN
	    #last_lay := false;
	END_IF;
	
	
	StartAutomat:
	CASE #_State OF
	    #STATE_INIT:
	        #CMD_On := FALSE;
	        #CMD_Mid := TRUE;
	        #CMD_Off := False;
	        
	        #CMD_OpenLodems := FALSE;
	        
	        #s_busy := FALSE;
	        #down_working := FALSE;
	        
	        #last_lay := FALSE;
	        #layer_holded := 0;
	        
	        #make_gasket_layer := FALSE;
	        
	        #_State := #STATE_AWAIT;
	        
	    #STATE_AWAIT:
	        #CMD_On := FALSE;
	        #CMD_Mid := TRUE;
	        #CMD_Off := False;
	        
	        // блокировки механизмов
	        #lock_forks := FALSE;
	        #lock_carousel := FALSE;
	        
	        #CMD_OpenLodems := NOT #ramp_not_down;
	        
	        #down_working := False;
	        
	        #sig_carousel_release_gaskets := false;
	        
	        #s_lay_cmd_permission := TRUE;
	        
	        // пушим пакет
	        IF (#push_packet) THEN
	            #_State := #STATE_PUSHING_PACKET;
	            GOTO EndAutomat;
	        END_IF;
	        
	        
	        IF (#s_busy) THEN
	            IF (#pick_gaskets AND #forks_start_sensor) THEN
	                #_State := #STATE_RELEASE_GASKETS;
	            #lock_forks := TRUE;
	            END_IF;
	        ELSE
	            
	            IF (#gaskets_acquire) THEN
	                #_State := #STATE_ACQUIRE_GASKETS;
	                #lock_carousel := TRUE;
	            ELSE
	                ;
	            END_IF;
	            
	        END_IF;
	        
	        
	    #STATE_RELEASE_GASKETS:
	        
	        #CMD_On := FALSE;
	        #CMD_Mid := FALSE;
	        #CMD_Off := #forks_start_sensor;
	        
	        #CMD_OpenLodems := FALSE;
	        
	        #down_working := TRUE;
	        
	        IF (#low_sensor) THEN
	            #_State := #STATE_OPENING_LODEMS;
	        END_IF;
	            
	    #STATE_OPENING_LODEMS:
	        #CMD_On := FALSE;
	        #CMD_Mid := FALSE;
	        #CMD_Off := TRUE;
	        
	        #CMD_OpenLodems := TRUE;
	        
	        #down_working := True;
	        
	        IF (#open_lodems_sensor AND #low_sensor) THEN
	            // ложементы свободны
	            #s_busy := FALSE;
	            
	            #_State := #STATE_AWAIT;
	        END_IF;
	        
	     
	    #STATE_ACQUIRE_GASKETS:
	            
	        #CMD_On := TRUE;
	        #CMD_Mid := FALSE;
	        #CMD_Off := False;
	        #CMD_OpenLodems := NOT #ramp_not_down;
	        
	        #lock_carousel := true;
	        
	        #s_lay_cmd_permission := FALSE;
	            
	        IF (NOT #gaskets_acquire) THEN
	            // если пропал до отдачи сигнала готовности значит был сброс или ошибка
	            //снимаемся с задачи
	            #_State := #STATE_AWAIT;
	            GOTO EndAutomat;
	        END_IF;
	        
	        // более надежный флаг поднятия каретки
	        IF (#top_sensor AND #top_sensor_filter) THEN
	            #_State := #STATE_WAIT_RELEASE;
	            #sig_carousel_release_gaskets := TRUE;
	        END_IF;
	        
	    #STATE_WAIT_RELEASE:
	        // как точно доехали наверх можем давать сигнал карусели об отдаче прокладок
	        #CMD_On := TRUE;
	        #CMD_Mid := FALSE;
	        #CMD_Off := False;
	        #CMD_OpenLodems := FALSE;
	        
	        #lock_carousel := FALSE;
	        
	        #sig_carousel_release_gaskets := TRUE;
	        
	        IF (#gaskets_released) THEN
	            #s_busy := TRUE;
	            #layer_holded := #layer_holded + 1;
	            
	            // решаем, надо ли еще слой прокладок положить
	            // TODO
	            // 
	            #last_lay := #layer_holded >= #QPLanksLayers - 1;
	            
	            #_State := #STATE_AWAIT;
	            GOTO EndAutomat;
	        END_IF;
	        
	        
	        IF (NOT #gaskets_busy) THEN
	            #_State := #STATE_AWAIT;
	            
	        END_IF;
	        
	    #STATE_PUSHING_PACKET:
	        
	        #s_lay_cmd_permission := FALSE;
	        
	        IF (NOT #s_busy AND (#gaskets_acquire OR NOT #gaskets_busy)) THEN
	            #CMD_On := TRUE;
	            #CMD_Mid := FALSE;
	            #CMD_Off := False;
	            
	            #CMD_OpenLodems := FALSE;
	            
	            // full reset carousel
	            // 
	            #carousel_full_reset := TRUE;
	            
	        END_IF;
	        
